IF reset THEN
	_bRetry := TRUE;
	Error 	:= FALSE;
	Aborted := FALSE;
END_IF

//============= State Control==================
IF NOT Execute THEN
	eSTATE:=STATE_RESETTING;
END_IF
IF Execute AND _bRetry AND NOT Robot._DI1.Error AND NOT Robot.Halt THEN
	PreviousStrStatus := strStatus;
	PreviousErrorCode := _UniqueErrorCode;
	uiExecutingStep   := uiResumeStep;
	Status := '';
	IF GVL_ADS.MachineState <>E_MachineState.Error THEN
		eSTATE:=STATE_EXECUTING;
	END_IF
END_IF
END_METHOD

METHOD  M_STATE_ABORTING
VAR_INPUT
END_VAR
CASE uiAbortingStep OF
	0 :
			
			tonTimeOut.IN 				:= FALSE;
			tonCheckRoundBeltDelay.IN	:= FALSE;
			_Abort := FALSE;
			_bRetry:= FALSE;
			IF strStatus = PreviousStrStatus THEN
				_UniqueErrorCode :=PreviousErrorCode;
			END_IF
			
			uiAbortingStep := 100;
    100:
			IF Robot._DI1.Error THEN
				uiAbortingStep := 200;
			ELSE
				uiAbortingStep := 9999;
			END_IF
	200:		
			 IF DAS_CoreSys.MachineControl.M_RobotResetCmd() THEN
				 uiAbortingStep := 300;
			 END_IF
	300:
			IF DAS_CoreSys.MachineControl.M_RobotStartCmd() THEN
				 uiAbortingStep := 400;
			 END_IF 
	400:
			IF Robot._DI1.Error THEN
		 		uiAbortingStep := 200;
			ELSE
				uiAbortingStep := 9999;
			END_IF
	9999:	
			_AbortCompleted:=TRUE;
END_CASE

IF _AbortCompleted THEN	
	eSTATE :=STATE_ABORTED;
END_IF
END_METHOD

METHOD  M_STATE_DONE
VAR_INPUT
END_VAR
Busy   := FALSE;
_Error := Error := FALSE;
_Abort := Abort := FALSE;
Done   := TRUE;

IF NOT Execute THEN
    eState := STATE_RESETTING;
END_IF
END_METHOD

METHOD  M_STATE_DORMANT
VAR_INPUT
END_VAR
// Clear FB output
Busy            := FALSE;
Done            := FALSE;
Aborted         := FALSE;
Error           := FALSE;
ErrorID         := 0;
Status          := '';
_ResetCompleted := FALSE;
_Error          := FALSE;
_Executed       := FALSE;

tonTimeOut.IN:=tonCheckRoundBeltDelay.IN:= FALSE;
strStatus :='FB_RobotRegionMove_RoundBelt: No Error';
uiExecutingStep :=uiResettingStep :=uiResumeStep :=0;
PreviousStrStatus			 :='';
PreviousErrorCode			 :='';
_bRetry			:= FALSE;
uiAbortingStep  := 0;
_AbortCompleted := FALSE;

// Wait Execute command
IF Execute AND NOT stop THEN
    eState := STATE_EXECUTING;
END_IF
END_METHOD

METHOD  M_STATE_ERROR
VAR_INPUT
END_VAR
ERROR   :=TRUE;
Busy	:=FALSE;
Status := strStatus;
UniqueErrorCode:=_UniqueErrorCode;
IF NOT Execute THEN	
eSTATE:=STATE_RESETTING;
END_IF
END_METHOD

METHOD  M_STATE_EXECUTING
VAR_INPUT
END_VAR
VAR_INST
	BoxReady_1st : BOOL;
	BoxReady_2nd : BOOL;
    uiBothStep : UINT;
    uiSingleClampStep : UINT;	
	Address_A : INT;
	Address_B : INT;
	A1Used	 : BOOL;
	A2Used	 : BOOL;
END_VAR
VAR
	
	
END_VAR
//20250418 note: current behavior : wait round belt finish rotating then check if box is ready , everything ready then call Robot start move
//				 Todo : consider if better call robot start move to waiting position and check box at same moment , Albert 

// Set Busy active edit by johnson
Busy := TRUE;
IF THIS^.Stop THEN // Pending the timeout when Stop signal occur
	tonTimeout.IN :=FALSE;
END_IF
// Service Process
CASE uiExecutingStep OF
	0:
        // Clear variable      
        uiBothStep := 0;
		uiSingleClampStep :=0;
		BoxReady_1st := 0;
		BoxReady_2nd := 0;
		tonTimeOut.IN:=FALSE;
		tonCheckRoundBeltDelay.IN :=FALSE;
        // Check command
        IF M_CheckCommand() THEN
            uiExecutingStep := 10;
		ELSE
			_Error:=TRUE;
        END_IF
    10:
        // Start process, check units first
        IF M_CheckUnitsReady() THEN
            uiExecutingStep := 20;
        END_IF
    20:
        // CHeck units not busy state
        IF M_CheckUnitsNotBusy() THEN
            uiExecutingStep := 30;
        END_IF
	30:
		IF M_CheckClampStatus() THEN
			uiExecutingStep := 1000;
		ELSE
			_Abort := TRUE;
		END_IF
   
	1000:   
			// Read   coordinate
			 Area := THIS^.Area;
 			 Address_A := LREAL_TO_INT(Info.A_Position);
			 Address_B := LREAL_TO_INT(Info.B_Position);
			 uiExecutingStep := 1100; 		
			 
	1100:
			// Check clamp userage
			IF UseA AND NOT UseB THEN
				//Only clampA
				A1Used := FALSE;
				A2Used := FALSE;
				uiExecutingStep := 10000;
			ELSIF NOT UseA AND UseB THEN
				//Only ClampB
				A1Used := FALSE;
				A2Used := FALSE;
				uiExecutingStep := 20000;
			ELSIF UseA AND UseB THEN
				//Both Clamps
				A1Used := TRUE;
				A2Used := TRUE;
				uiExecutingStep := 30000;
			END_IF
       
    10000: // Only ClampA 
        IF NOT Robot._DI1.Done THEN
			// Delay to make sure round belt is starting/finish rotating
			IF NOT RoundBelt.xBusy AND NOT RoundBelt.xError THEN
				tonCheckRoundBeltDelay.IN:=TRUE;
			ELSE
				tonCheckRoundBeltDelay.IN:=FALSE;	
			END_IF
		
		
		CASE uiSingleClampStep OF
			0:
				CASE Address_A OF						
							1: A1Used := TRUE;
							2: A2Used := TRUE;
				END_CASE
				
				IF tonCheckRoundBeltDelay.Q THEN
					 uiSingleClampStep:=50;  
				END_IF
				
			50:
				IF Get THEN  // Picking job , check box is ready
					IF A1Used AND Input.bRoundBelt_ChangeZoneA2Detect_Sensor =FALSE	THEN
						uiResettingStep := 10000;
						_Abort:=TRUE	;
						strStatus :='FB_RobotRegionMove_RoundBelt Step 10000: No Box on A1';
					ELSIF A2Used AND Input.bRoundBelt_ChangeZoneA3Detect_Sensor =FALSE	THEN
						uiResettingStep := 10000;
						_Abort:=TRUE	;
						strStatus :='FB_RobotRegionMove_RoundBelt Step 10000: No Box on A2';
					ELSE 
						uiSingleClampStep := 100;
					END_IF	
				ELSE		//Place job , check no box 
					IF A1Used AND Input.bRoundBelt_ChangeZoneA2Detect_Sensor =TRUE	THEN
						uiResettingStep := 10000;
						_Abort:=TRUE	;
						strStatus :='FB_RobotRegionMove_RoundBelt Step 10000: Box on A1';									
					ELSIF A2Used AND Input.bRoundBelt_ChangeZoneA3Detect_Sensor =TRUE	THEN
						uiResettingStep := 10000;
						_Abort:=TRUE	;
						strStatus :='FB_RobotRegionMove_RoundBelt Step 10000: Box on A2';
					ELSE
						uiSingleClampStep := 100;	
					END_IF				
				END_IF
	  
		  100 :  
		  		IF get THEN
					BoxReady_1st := (A1Used AND Input.bRoundBelt_ChangeZoneA2Detect_Sensor) OR
		  						 (A2Used AND Input.bRoundBelt_ChangeZoneA3Detect_Sensor);
				ELSE
					BoxReady_1st := (A1Used AND NOT Input.bRoundBelt_ChangeZoneA2Detect_Sensor) OR
		  						 (A2Used AND NOT Input.bRoundBelt_ChangeZoneA3Detect_Sensor);
				END_IF		
				IF BoxReady_1st THEN
					uiSingleClampStep:=9999;  
				END_IF			 
								 
		  9999:// 
	
		END_CASE				          		 
				  // Robot Abs move
           		 Robot.M_StartRobotAbsMove(GetBox:=Get,
											UseClampA:=UseA,
											UseClampB:=UseB,
											Area:=Area,
											ClampA_Address:=Address_A,
											ClampB_Address:=Address_B,
											BoxReady_1:=BoxReady_1st,
											BoxReady_2:=BoxReady_2nd);				  
		
        ELSE
			tonTimeOut.IN:=FALSE;
            uiExecutingStep := 10080;
        END_IF
			tonTimeOut.IN:=TRUE;
		IF tonTimeOut.Q=TRUE THEN
			uiResumeStep 	:= 10000;
			tonTimeOut.IN	:= FALSE;
			strStatus := 'FB_RobotRegionMove_RoundBelt Step 10000: Robot Abs Move timeout';
			_Abort			:= TRUE;
		END_IF	
		IF robot.Error THEN
			uiResumeStep 	:= 10000;
			tonTimeOut.IN	:= FALSE;
			_Abort 			:= TRUE;
			strStatus := CONCAT('FB_RobotRegionMove_RoundBlet Step 10000 : ',robot.ErrMsg);
		END_IF
    10080:
        Robot.M_ResetRobotAbsMove(UseA,UseB); // Clear command and go to place box
		tonTimeOut.IN:=TRUE;
        IF NOT Robot._DI1.Done THEN
			tonTimeOut.IN:=FALSE;
            uiExecutingStep := 99000; 
        END_IF
    	IF tonTimeOut.Q=TRUE THEN
			strStatus :='FB_RobotRegionMove_RoundBelt Step 10080: Reset Robot timeout';


			_Error:=TRUE;
		END_IF	
    
   20000: // Only ClampB
        IF NOT Robot._DI1.Done THEN
           IF NOT RoundBelt.xBusy AND NOT RoundBelt.xError THEN
				tonCheckRoundBeltDelay.IN:=TRUE;
			ELSE
				tonCheckRoundBeltDelay.IN:=FALSE;	
			END_IF
		
		
		CASE uiSingleClampStep OF
			0:
				CASE Address_B OF						
							1: A1Used := TRUE;
							2: A2Used := TRUE;
				END_CASE
				
				IF tonCheckRoundBeltDelay.Q THEN
					 uiSingleClampStep:=50;  
				END_IF
			
			50: 
				IF Get THEN  // Picking job , check box is ready
					IF A1Used AND Input.bRoundBelt_ChangeZoneA2Detect_Sensor =FALSE	THEN
						_Abort:=TRUE	;
						uiResettingStep := 20000;
						strStatus :='FB_RobotRegionMove_RoundBelt Step 20000: No Box on A1';		
					ELSIF A2Used AND Input.bRoundBelt_ChangeZoneA3Detect_Sensor =FALSE	THEN
						_Abort:=TRUE	;
						uiResettingStep := 20000;
						strStatus :='FB_RobotRegionMove_RoundBelt Step 20000: No Box on A2';
					ELSE
						uiSingleClampStep := 100;
					END_IF	
				ELSE		//Place job , check no box 
					IF A1Used AND Input.bRoundBelt_ChangeZoneA2Detect_Sensor =TRUE	THEN
						_Abort:=TRUE	;
						uiResettingStep := 20000;
						strStatus :='FB_RobotRegionMove_RoundBelt Step 20000: Box on A1';				
					ELSIF A2Used AND Input.bRoundBelt_ChangeZoneA3Detect_Sensor =TRUE	THEN
						_Abort:=TRUE	;
						uiResettingStep := 20000;
						strStatus :='FB_RobotRegionMove_RoundBelt Step 20000: Box on A2';
					ELSE
						uiSingleClampStep := 100;
					END_IF				
				END_IF
	  
		  100 :  
		  		IF get THEN
					BoxReady_2nd := (A1Used AND Input.bRoundBelt_ChangeZoneA2Detect_Sensor) OR
		  						 (A2Used AND Input.bRoundBelt_ChangeZoneA3Detect_Sensor);
				ELSE
					BoxReady_2nd := (A1Used AND NOT Input.bRoundBelt_ChangeZoneA2Detect_Sensor) OR
		  						 (A2Used AND NOT Input.bRoundBelt_ChangeZoneA3Detect_Sensor);
				END_IF		
				IF BoxReady_2nd THEN
					uiSingleClampStep:=9999;  
				END_IF			 
								 
		  9999:// 
	
		END_CASE				          		 
					  // Robot Abs move
           		 Robot.M_StartRobotAbsMove( GetBox:=Get,
											UseClampA:=UseA,
											UseClampB:=UseB,
											Area:=Area,
											ClampA_Address:=Address_A,
											ClampB_Address:=Address_B,
											BoxReady_1:=BoxReady_1st,
											BoxReady_2:=BoxReady_2nd);		  
		
        ELSE
			tonTimeOut.IN:=FALSE;
            uiExecutingStep := 20080;
        END_IF	
		tonTimeOut.IN:=TRUE;
		IF tonTimeOut.Q=TRUE THEN
			uiResumeStep 	:= 20000;
			tonTimeOut.IN	:= FALSE;
			strStatus := 'FB_RobotRegionMove_RoundBelt Step 20000: Robot Abs Move timeout';
			_Abort			:= TRUE;
		END_IF
		IF robot.Error THEN
			uiResumeStep := 20000;
			_Abort := TRUE;
			strStatus := CONCAT('FB_RobotRegionMove_RoundBlet Step 20000 : ',robot.ErrMsg);
		END_IF		          		 
			
       
		
    20080:
       Robot.M_ResetRobotAbsMove(UseA,UseB);; // Clear command
		tonTimeOut.IN:=TRUE;
        IF NOT Robot._DI1.Done THEN
			tonTimeOut.IN:=FALSE;
            uiExecutingStep := 99000;
        END_IF
		IF tonTimeOut.Q=TRUE THEN
			strStatus :='FB_RobotRegionMove_RoundBelt Step 20080: Reset Robot timeout';


			_Error:=TRUE;
		END_IF	
    30000: // Both Clamps
        	
			IF NOT RoundBelt.xBusy AND NOT RoundBelt.xError THEN
				tonCheckRoundBeltDelay.IN:=TRUE;
			ELSE
				tonCheckRoundBeltDelay.IN:=FALSE;	
			END_IF
		
		  CASE uiBothStep OF
           		0://	
					BoxReady_1st := FALSE;
					BoxReady_2nd := FALSE;
					
					IF tonCheckRoundBeltDelay.Q THEN
						uiBothStep:=100;	
					END_IF
				100:
					IF Get THEN  // Picking job , check box is ready
						IF  Input.bRoundBelt_ChangeZoneA2Detect_Sensor =FALSE	THEN
							_Abort:=TRUE	;
							uiResettingStep := 30000;
							strStatus :='FB_RobotRegionMove_RoundBelt Step 30000: No Box on A1';
						END_IF				
						IF  Input.bRoundBelt_ChangeZoneA3Detect_Sensor =FALSE	THEN
							_Abort:=TRUE	;
							uiResettingStep := 30000;
							strStatus :='FB_RobotRegionMove_RoundBelt Step 30000: No Box on A2';
						END_IF	
					ELSE		//Place job , check no box 
						IF  Input.bRoundBelt_ChangeZoneA2Detect_Sensor =TRUE	THEN
							_Abort:=TRUE	;
							uiResettingStep := 30000;
							strStatus :='FB_RobotRegionMove_RoundBelt Step 30000: Box on A1';
						END_IF				
						IF  Input.bRoundBelt_ChangeZoneA3Detect_Sensor =TRUE	THEN
							_Abort:=TRUE	;
							uiResettingStep := 30000;
							strStatus :='FB_RobotRegionMove_RoundBelt Step 30000: Box on A2';
						END_IF				
					END_IF
					IF NOT _Error THEN
						uiBothStep:=1000;
					END_IF
				1000:	
						
						BoxReady_1st :=TRUE;
						uiBothStep:=2000;
					
						
				2000:					
						IF Robot._DI1.Notification THEN
							uiBothStep:=3000;
						END_IF
				3000:	
						 BoxReady_2nd :=TRUE;						 
					     uiBothStep:=9999;
				
				9999: //Wait		
        // wait reset
        END_CASE

       	  // Robot Abs move
           		 Robot.M_StartRobotAbsMove( GetBox:=Get,
											UseClampA:=UseA,
											UseClampB:=UseB,
											Area:=Area,
											ClampA_Address:=Address_A,
											ClampB_Address:=Address_B,
											BoxReady_1:=BoxReady_1st,
											BoxReady_2:=BoxReady_2nd);	
		
		
        IF Robot._DI1.Done THEN
			tonTimeOut.IN:=FALSE;
            uiExecutingStep := 30080;
        END_IF
		tonTimeOut.IN:=TRUE;
		IF tonTimeOut.Q=TRUE THEN
			uiResumeStep 	:= 30000;
			tonTimeOut.IN	:= FALSE;
			strStatus := 'FB_RobotRegionMove_RoundBelt Step 30000: Robot Abs Move timeout';
			_Abort			:= TRUE;
		END_IF
		IF robot.Error THEN
			uiResumeStep := 30000;
			_Abort := TRUE;
			strStatus := CONCAT('FB_RobotRegionMove_RoundBlet Step 30000 : ',Robot.ErrMsg);
		END_IF	
		
    30080: // Check robot command is clear
        
        Robot.M_ResetRobotAbsMove(UseA,UseB);

        IF NOT Robot._DI1.Done THEN
			tonTimeOut.IN:=FALSE;
            uiExecutingStep := 99000; // go to place step
        END_IF    
   		tonTimeOut.IN:=TRUE;
		IF tonTimeOut.Q=TRUE THEN
			strStatus :='FB_RobotRegionMove_RoundBelt Step 30080: Stop Robot timeout';




			_Error:=TRUE;
		END_IF	
   
    99000:
			IF Get THEN  // Picking job , check box putted
				IF A1Used AND Input.bRoundBelt_ChangeZoneA2Detect_Sensor =TRUE	THEN
					_Error:=TRUE	;
					strStatus :='FB_RobotRegionMove_RoundBelt Step 99000: Box still on A1';


				END_IF				
				IF A2Used AND Input.bRoundBelt_ChangeZoneA3Detect_Sensor =TRUE	THEN
					_Error:=TRUE	;
					strStatus :='FB_RobotRegionMove_RoundBelt Step 99000: Box still on A2';


				END_IF	
			ELSE		//Place job , check no box 
				IF A1Used AND Input.bRoundBelt_ChangeZoneA2Detect_Sensor =FALSE	THEN
					_Error:=TRUE	;
					strStatus :='FB_RobotRegionMove_RoundBelt Step 99000: No Box on A1';


				END_IF				
				IF A2Used AND Input.bRoundBelt_ChangeZoneA3Detect_Sensor =FALSE	THEN
					_Error:=TRUE	;
					strStatus :='FB_RobotRegionMove_RoundBelt Step 99000: No Box on A2';


				END_IF	
			
			END_IF
			IF NOT _Error THEN
			 	uiExecutingStep := 99100;
			 END_IF
	99100: // process done
                Status    := 'FB_RobotRegionMove_RoundBelt Step 99100: Process completed';
        	_Executed := TRUE;
END_CASE

// ==================== STATE Control ========================
IF NOT Execute THEN
    eState 	:= STATE_RESETTING;
ELSIF _Error THEN
    eState 	:= STATE_ERROR;
ELSIF _Abort THEN
	eSTATE	:= STATE_ABORTING;
ELSIF _Executed THEN
    eState 	:= STATE_DONE;
END_IF
END_METHOD

METHOD  M_STATE_RESETTING
VAR_INPUT
END_VAR
// Done := false 更改到Dormant 清除確保，上位檢查到done 後可以直接下Execute

CASE uiResettingStep OF

	0:
		tonTimeOut.IN:=FALSE;
		Robot.M_ResetAllCommand();
		Robot.M_ResetRobotAbsMove(TRUE,TRUE);
		uiResettingStep:=100;

	100:

		uiResettingStep:=9999;
		
	9999:
//		Done := FALSE;
//		Busy := FALSE;
		_ResetCompleted:=TRUE;
END_CASE
IF _ResetCompleted THEN
	eSTATE:=STATE_DORMANT;
END_IF
END_METHOD

END_FUNCTION_BLOCK

// ---- Library/20_MachineUnits/21_StorageArea/Service_Robot/FB_RobotAbsMove_V2.TcPOU
// Jidien Kachu Edited in 2025/10/14
FUNCTION_BLOCK FB_RobotAbsMove_V2 EXTENDS FB_ObjectBase_V2 IMPLEMENTS IBasicElement
VAR_INPUT
    Robot         				: REFERENCE TO FB_FanucRobot_Basic_V2;
    LowerConveyor 				: REFERENCE TO FB_Motor;
    // Command   : ST_WareHouseWithRobotMove_Command;
    Info 						: st_AutoSixAxisAbsMoveParameter;
	Input 						: ST_InputTable;
    Stop 						: BOOL;
	Output 						: ST_OutputTable;
	Cylinder 					: REFERENCE TO UNI_CylinderList;
	bCheckUpperCV_ServiceDone	: BOOL;
END_VAR
VAR_OUTPUT
    // Status : ST_WareHouseWithRobotMove_Status;
	AClampMoveDone	: BOOL;
	BClampMoveDone	: BOOL;
END_VAR
VAR
    //_Abort       : BOOL;
    strStatus    : STRING;
    uiResumeStep : UINT;

    Area : E_RobotArea;
    UseA : BOOL;
    UseB : BOOL;

    Get                         : BOOL;
    tonTimeOut                  : TON;
	bTimeOutIN					: BOOL;
	tonDelay					 : TON;
    _UniqueErrorCode            : STRING;
    FirstSensorOfLowerConveyor  : BOOL;
    SecondSensorOfLowerConveyor : BOOL;

	//Added by Jidien Kachu in 2025/10/09
	uiLastBothStep	: UINT;
	uiLastSingleClampStep	: UINT;
	bRobotTimeOutIN	: BOOL;
	tonRobotTimeOut	: TON;
	uiBothStep	: UINT;
	uiSingleClampStep	: UINT;
	bMotorDelayIN	: BOOL;
	tonMotorDelay	: TON;
	bIOTimeoutIN	: BOOL;
	tonIOTimeout	: TON;
	bRetry: BOOL;
	
	//Added by Gamin in 2025//11/24
	_AClampDoingWork	: BOOL;
	_BClampDoingWork	: BOOL;
END_VAR

SUPER^.A10_StateControl();
A00_BasicUnits();
FirstSensorOfLowerConveyor := Input.bLowCV_BoxArrived_Sensor;
SecondSensorOfLowerConveyor := NOT Input.bLowCV_2ndBoxGap_Sensor;// .bLowCV_Block2Detect_Sensor;

(*============================================================
Create Date : 2025/11/22
Last Update	: 2026/04/01
Change Log  : 2025/11/24，send flag A clamp done and B clamp done for C# use to SQL // Edited : Gamin
			  2026/04/01，移植泰興鏡射機版本。
============================================================*)

ACTION A00_BasicUnits:
tonTimeOut(IN:= bTimeOutIN AND NOT THIS^.Stop, PT:=T#60S);
tonDelay(PT:=T#1S);
ErrorID :=2200;
tonMotorDelay(IN:= bMotorDelayIN,PT:=T#1S);
tonIOTimeout(IN:= bIOTimeoutIN,PT:= T#1S);
END_ACTION

METHOD M_CheckClampStatus : BOOL
VAR_INPUT
END_VAR
M_CheckClampStatus := FALSE;

IF NOT UseA AND NOT UseB THEN
	M_CheckClampStatus 	:= FALSE;
	strStatus 			:= 'FB_RobotAbsMove_V2: Wrong Command , Both Clammp not used';
	RETURN;
END_IF

IF UseA THEN
	IF Get THEN
		IF NOT Robot._DI1.ClampA_Open THEN
			M_CheckClampStatus  := FALSE;
			strStatus			:= 'FB_RobotAbsMove_V2: Robot Use A Clamp Get ,but Clamp not open ';
			RETURN;
		END_IF
	ELSE
		IF Robot._DI1.ClampA_Open THEN
			M_CheckClampStatus	:= FALSE;
			strStatus			:= 'FB_RobotAbsMove_V2: Robot Use A Clamp Place ,but Clamp open';
			RETURN;
		END_IF
	END_IF
END_IF
IF UseB THEN
	IF Get THEN
		IF NOT Robot._DI1.ClampB_Open THEN
			M_CheckClampStatus  := FALSE;
			strStatus			:= 'FB_RobotAbsMove_V2: Robot Use B Clamp Get ,but Clamp not open ';
			RETURN;
		END_IF
	ELSE
		IF Robot._DI1.ClampB_Open THEN
			M_CheckClampStatus	:= FALSE;
			strStatus			:= 'FB_RobotAbsMove_V2: Robot Use B Clamp Place ,but Clamp open';
			RETURN;
		END_IF
	END_IF
END_IF

M_CheckClampStatus := TRUE;
END_METHOD

METHOD M_CheckCommand : BOOL // True : Command is useful
VAR_INPUT
END_VAR
VAR
	
END_VAR
// Check command paremeter is correct


IF Info.A_Get <> Info.B_Get THEN
	strStatus:='FB_RobotAbsMove_V2: Wrong command ,GetA not match to GetB';
	M_CheckCommand:=FALSE;
	RETURN;
ELSE		
	THIS^.Get :=Info.A_Get;
END_IF

IF Info.A_Area<> Info.B_Area THEN
	IF NOT(Info.A_Area=99 OR Info.B_Area=99) THEN
	strStatus:='FB_RobotAbsMove_V2: Wrong command ,Area A not match to Area B';
	M_CheckCommand:=FALSE;
	RETURN;
END_IF
END_IF

IF Info.A_Area = 99 AND Info.B_Area = 99 THEN
	strStatus:='FB_RobotAbsMove_V2: Wrong command ,Both Area are 99';
	M_CheckCommand:=FALSE;
	RETURN;
END_IF

CASE LREAL_TO_INT(Info.A_Area) OF
	1 : //Normal command : RoundBelt
		IF Info.A_Position<1 OR  Info.A_Position>3 THEN
			strStatus:='FB_RobotAbsMove_V2: Wrong command ,Position A Not allow';
			M_CheckCommand:=FALSE;
			RETURN;	
		ELSE
			Area := E_RobotArea.RoundBelt;
			UseA :=TRUE	;	
		END_IF
		
	2:	//Buffer area
		IF Info.A_Position<1 OR  Info.A_Position>40 THEN
			strStatus:='FB_RobotAbsMove_V2: Wrong command ,Position A Not allow';
			M_CheckCommand:=FALSE;
			RETURN;	
		ELSE
			Area := E_RobotArea.BufferArea;
			UseA :=TRUE	;	
		END_IF
	3: //Allocated/Empty conveyor
		IF Info.A_Position<1 OR  Info.A_Position>2 THEN
			strStatus:='FB_RobotAbsMove_V2: Wrong command ,Position A Not allow';
			M_CheckCommand:=FALSE;
			RETURN;	
		ELSE
			Area := E_RobotArea.TransmitCV;
			UseA :=TRUE	;	
		END_IF
	5: //FeedIn/Out conveyor
		IF Info.A_Position<1 OR  Info.A_Position>5 THEN
			strStatus:='FB_RobotAbsMove_V2: Wrong command ,Position A Not allow';
			M_CheckCommand:=FALSE;
			RETURN;	
		ELSIF Info.A_Position=3 AND Get THEN
			strStatus:='FB_RobotAbsMove_V2: Wrong command ,Can Not Get box from FeedOut conveyor ';
			M_CheckCommand:=FALSE;
			RETURN;	
		ELSE
			Area := E_RobotArea.InOutConveyor;
			UseA :=TRUE	;	
		END_IF
	7: // PullOut conveyor
		IF Info.A_Position<1 OR  Info.A_Position>2 THEN
			strStatus:='FB_RobotAbsMove_V2: Wrong command ,Position A Not allow';
			M_CheckCommand:=FALSE;
			RETURN;	
		ELSE
			Area := E_RobotArea.PullOutConveyor;
			UseA :=TRUE	;	
		END_IF
	
	99: //ClampA not use
		UseA :=FALSE;
	
	ELSE //Wrong command
		strStatus:='FB_RobotAbsMove_V2: Wrong command ,Area_A not allow ';
		M_CheckCommand:=FALSE;
		RETURN;

END_CASE

CASE LREAL_TO_INT(Info.B_Area) OF
	1 : //Normal command : RoundBelt
		IF Info.B_Position<1 OR  Info.B_Position>3 THEN
			strStatus:='FB_RobotAbsMove_V2: Wrong command ,Position B Not allow';
			M_CheckCommand:=FALSE;
			RETURN;	
		ELSE
			Area := E_RobotArea.RoundBelt;
			UseB :=TRUE	;	
		END_IF
		
	2:	
		IF Info.B_Position<1 OR  Info.B_Position>40 THEN
			strStatus:='FB_RobotAbsMove_V2: Wrong command ,Position B Not allow';
			M_CheckCommand:=FALSE;
			RETURN;	
		ELSE
			Area := E_RobotArea.BufferArea;
			UseB :=TRUE	;	
		END_IF
	3:
		IF Info.B_Position<1 OR  Info.B_Position>2 THEN
			strStatus:='FB_RobotAbsMove_V2: Wrong command ,Position B Not allow';
			M_CheckCommand:=FALSE;
			RETURN;	
		ELSE
			Area := E_RobotArea.TransmitCV;
			UseB :=TRUE	;	
		END_IF
	5:
		IF Info.B_Position<1 OR  Info.B_Position>5 THEN
			strStatus:='FB_RobotAbsMove_V2: Wrong command ,Position B Not allow';
			M_CheckCommand:=FALSE;
			RETURN;	
		ELSE
			Area := E_RobotArea.InOutConveyor;
			UseB :=TRUE	;	
		END_IF
	7:
		IF Info.B_Position<1 OR  Info.B_Position>2 THEN
			strStatus:='FB_RobotAbsMove_V2: Wrong command ,Position B Not allow';
			M_CheckCommand:=FALSE;
			RETURN;	
		ELSIF Info.B_Position=3 AND Get THEN
			strStatus:='FB_RobotAbsMove_V2: Wrong command ,Can Not Get box from FeedOut conveyor ';
			M_CheckCommand:=FALSE;
			RETURN;	
		ELSE
			Area := E_RobotArea.PullOutConveyor;
			UseB :=TRUE	;	
		END_IF
	
	99: //ClampA not use
		UseB :=FALSE;
	
	ELSE //Wrong command
		strStatus:='FB_RobotAbsMove_V2: Wrong command ,Area_B not allow ';
		M_CheckCommand:=FALSE;
		RETURN;

END_CASE


M_CheckCommand:=TRUE;
END_METHOD

METHOD M_CheckUnitsNotBusy : BOOL
VAR_INPUT
END_VAR
M_CheckUnitsNotBusy := true;
END_METHOD

METHOD M_CheckUnitsReady : BOOL
VAR_INPUT
END_VAR
M_CheckUnitsReady := true;
END_METHOD

METHOD  M_STATE_ABORTED
VAR_INPUT
END_VAR

//Edited by Jidien Kachu in 2025/10/28
IF NOT bRetry THEN
	ERROR :=TRUE;
	Busy    := FALSE;
	Aborted := TRUE;
	Status := strStatus;
	UniqueErrorCode:=_UniqueErrorCode;
	uiAbortingStep := 0;
	_AbortCompleted:=FALSE;//Edited by Jidien Kachu in 2025/10/14
END_IF

IF Reset THEN
	bRetry := TRUE;
	ERROR :=FALSE;
	Aborted := FALSE;
END_IF
IF NOT Execute THEN
	eSTATE:=STATE_RESETTING;
END_IF

IF Execute AND bRetry AND NOT Robot.Error AND NOT Robot.Halt THEN
	uiExecutingStep :=uiResumeStep;

	//Edited by Jidien Kachu in 2025/10/14
	uiBothStep := uiLastBothStep;
	uiSingleClampStep := uiLastSingleClampStep;
	Status := '';


	//////////////////////////////////////
	IF GVL_ADS.MachineState <>E_MachineState.Error THEN
		eSTATE:=STATE_EXECUTING;
	END_IF
END_IF
END_METHOD

METHOD  M_STATE_ABORTING
VAR_INPUT
END_VAR
CASE uiAbortingStep OF
	0 :
			tonDelay.IN 	   := FALSE;
			bTimeOutIN  	   := FALSE;
			tonRobotTimeOut.IN := FALSE;
			_Abort 			   := FALSE;
			bRetry			   := FALSE;
			//Edited by Jidien Kachu in 2025/10/14
			LowerConveyor.M_MotorStop();
			IF 	LowerConveyor.InStopped THEN
				uiAbortingStep:=100;
			END_IF
    100:
			IF Robot._DI1.Error THEN
				uiAbortingStep := 200;
			ELSE
				uiAbortingStep := 9999;
			END_IF
	200:		
			 IF DAS_CoreSys.MachineControl.M_RobotResetCmd() THEN
				 uiAbortingStep := 300;
			 END_IF
	300:
			IF DAS_CoreSys.MachineControl.M_RobotStartCmd() THEN
				 uiAbortingStep := 400;
			 END_IF 
	400:
			IF Robot._DI1.Error THEN
		 		uiAbortingStep := 200;
			ELSE
				uiAbortingStep := 9999;
			END_IF
	
	9999:	
			_AbortCompleted:=TRUE;
END_CASE

IF _AbortCompleted THEN	
	eSTATE :=STATE_ABORTED;
END_IF
END_METHOD

METHOD  M_STATE_DONE
VAR_INPUT
END_VAR
Busy   := FALSE;
_Error := Error := FALSE;
_Abort := Abort := FALSE;
Done   := TRUE;

IF NOT Execute THEN
    eState := STATE_RESETTING;
END_IF
END_METHOD

METHOD  M_STATE_DORMANT
VAR_INPUT
END_VAR
// Clear FB output
Busy            := FALSE;
Done            := FALSE;
Aborted         := FALSE;
Error           := FALSE;
ErrorID         := 0;
Status          := '';
_ResetCompleted := FALSE;
_AbortCompleted := FALSE;
_Error          := FALSE;
_Executed       := FALSE;
tonDelay.IN := FALSE	;
bTimeOutIN:=FALSE;
strStatus :='FB_RobotAbsMove_V2: No Error';
uiExecutingStep :=uiResettingStep :=uiResumeStep :=0;
AClampMoveDone	:= FALSE;
BClampMoveDone	:= FALSE;
_AClampDoingWork	:= FALSE;
_BClampDoingWork	:= FALSE;
bRetry := FALSE;
uiBothStep := 0;
uiSingleClampStep :=0;

// Wait Execute command
IF Execute AND NOT stop THEN
    eState := STATE_EXECUTING;
END_IF
END_METHOD

METHOD  M_STATE_ERROR
VAR_INPUT
END_VAR
ERROR   :=TRUE;
Busy	:=FALSE;
Status := strStatus;
UniqueErrorCode:=_UniqueErrorCode;
ErrorID :=2200;

IF NOT Execute THEN	
	eSTATE:=STATE_RESETTING;
END_IF
END_METHOD

METHOD  M_STATE_EXECUTING
VAR_INPUT
END_VAR
VAR_INST
    ActionMode       : E_ReloadRoundBoxAction;
	BoxReady_1st : BOOL;
	BoxReady_2nd : BOOL;
    CarrierReady_1st : BOOL;
    CarrierReady_2nd : BOOL;
    //uiBothStep : UINT;
    //uiSingleClampStep : UINT;	
	Area : E_RobotArea;
	Address_A : INT;
	Address_B : INT;
END_VAR
VAR
	WareHouse: INT;
END_VAR
// Set Busy active edit by johnson
Busy := TRUE;
(*IF THIS^.Stop THEN // Pending the timeout when Stop signal occur
	tonTimeout.IN :=FALSE;
END_IF*)
// Service Process
CASE uiExecutingStep OF
	0:
        // Clear variable
        ActionMode       := E_ReloadRoundBoxAction.Undefined;
        CarrierReady_1st := FALSE;
        CarrierReady_2nd := FALSE;
        uiBothStep := 0;
		uiSingleClampStep :=0;
		uiLastBothStep := 0;//Edited by Jidien Kachu in 2025/10/14
		uiLastSingleClampStep := 0;//Edited by Jidien Kachu in 2025/10/14
		BoxReady_1st := FALSE;
		BoxReady_2nd := FALSE;
		bTimeOutIN:=FALSE;
        // Check command
        IF M_CheckCommand() THEN
            uiExecutingStep := 10;
		ELSE
			_Error:=TRUE;
        END_IF
    10:
        // Start process, check units first
        IF M_CheckUnitsReady() THEN
            uiExecutingStep := 20;
        END_IF
    20:
        // CHeck units not busy state
        IF M_CheckUnitsNotBusy() THEN
            uiExecutingStep := 30;
        END_IF
	30:
		IF M_CheckClampStatus() THEN
            uiExecutingStep := 1000;
		ELSE
			_Abort := TRUE;
        END_IF
   
	1000:   
			// Read   coordinate
			 Area := THIS^.Area;
 			 Address_A := LREAL_TO_INT(Info.A_Position);
			 Address_B := LREAL_TO_INT(Info.B_Position);
			 
			IF UseA AND NOT UseB THEN
				//Only clampA
				uiExecutingStep := 10000;
			ELSIF NOT UseA AND UseB THEN
				//Only ClampB 
				uiExecutingStep := 20000;
			ELSIF UseA AND UseB THEN
				//Both Clamps
				uiExecutingStep := 30000;		
			END_IF
       
    10000: // Only ClampA 
        IF NOT Robot._DI1.Done THEN
            //Edited by Jidien Kachu in 2025/10/14
				CASE uiSingleClampStep OF
					0://
						IF Area= E_RobotArea.InOutConveyor AND Address_A=3 THEN
							IF Cylinder.List.fbLowCV_Block1.InRearPosition THEN
								uiSingleClampStep:=100;// Need to control feedout conveyor
							ELSE
								_Error := TRUE;
								strStatus := 'FB_RobotAbsMove_V2 Step 10000: Block 2 cylinder inrearPosition';
							END_IF
						ELSE
							uiSingleClampStep:=1000;	
						END_IF
					100:	
						tonDelay.IN := FALSE	;
						LowerConveyor.M_MoveBackward();
						IF (NOT FirstSensorOfLowerConveyor) AND (NOT SecondSensorOfLowerConveyor) THEN
							bTimeOutIN:=FALSE;;
							uiSingleClampStep:=150;
						END_IF
						bTimeOutIN:=TRUE;
						//Edited by Jidien Kachu in 2025/10/14
						IF tonTimeOut.Q=TRUE OR robot._DI1.Error THEN
							strStatus :='FB_RobotAbsMove_V2 Step 10000: Empty Conveyor timeout';
	//						_Error:=TRUE;
							_Abort := TRUE;
							uiLastSingleClampStep := 0;
							uiResumeStep := 10000;
							uiAbortingStep := 0;
						END_IF
						//////////////////////////////////////////
					150:
						tonDelay.IN := TRUE;
						IF tonDelay.Q THEN
							uiSingleClampStep:=200;
						END_IF	
					200:
						tonDelay.IN := FALSE	;
						LowerConveyor.M_MotorStop();
						uiSingleClampStep:=300;
					
					300:
						IF 	LowerConveyor.InStopped THEN
							bTimeOutIN:=FALSE;
							BoxReady_1st:=TRUE;
							uiSingleClampStep:=9999;
						END_IF
						bTimeOutIN:=TRUE;
						//Edited by Jidien Kachu in 2025/10/14
						IF tonTimeOut.Q=TRUE OR Robot._DI1.Error THEN
							strStatus :='FB_RobotAbsMove_V2 Step 10000: Stop Conveyor timeout';
	//						_Error:=TRUE;
							_Abort := TRUE;
							uiLastSingleClampStep := 200;
							uiResumeStep := 10000;
							uiAbortingStep := 0;
						END_IF	
						//////////////////////////////////////////
					1000:
						// 檢查 A爪去夾爪時，要確保上層輸送帶是完成的。
							IF Area= E_RobotArea.InOutConveyor AND Address_A = 2 THEN
								IF bCheckUpperCV_ServiceDone THEN
									BoxReady_1st:=TRUE;
									_AClampDoingWork := TRUE;
									uiSingleClampStep:=9999;
								END_IF
							ELSE
							BoxReady_1st:=TRUE;
							_AClampDoingWork := TRUE;
							uiSingleClampStep:=9999;
							END_IF
					9999: //Wait	
				END_CASE
//			END_IF
			
			          		 
				  // Robot Abs move
           		 Robot.M_StartRobotAbsMove(GetBox:=Get,
											UseClampA:=UseA,
											UseClampB:=UseB,
											Area:=Area,
											ClampA_Address:=Address_A,
											ClampB_Address:=Address_B,
											BoxReady_1:=BoxReady_1st,
											BoxReady_2:=BoxReady_2nd);		

			// robot doing AClamp done
			IF Get THEN
				IF _AClampDoingWork AND NOT Robot._DI1.ClampA_Open THEN
					AClampMoveDone := TRUE;
				END_IF
			ELSE
				IF _AClampDoingWork AND Robot._DI1.ClampA_Open THEN
					AClampMoveDone := TRUE;
				END_IF
			END_IF	  
		
        ELSE
            uiExecutingStep := 10080;
        END_IF
		IF tonRobotTimeOut.Q THEN
			_Abort 		 := TRUE;
			uiResumeStep := 10000;
			strStatus 	 := 'FB_RobotAbsMove_V2 Step 10000: Robot Move timeout';
		END_IF
		IF Robot._DI1.Error THEN
			_Abort		:= TRUE;
			uiResumeStep:= 10000;
			strStatus	:= CONCAT(STR1 := 'FB_RobotAbsMove_V2 Step 10000:',
								  STR2 := Robot.ErrMsg);
        END_IF
		
    10080:
        Robot.M_ResetRobotAbsMove(UseA,UseB); // Clear command and go to place box
		bTimeOutIN:=TRUE;
        IF NOT Robot._DI1.Done THEN
			bTimeOutIN:=FALSE;
            uiExecutingStep := 40000; 
        END_IF
    	IF tonTimeOut.Q=TRUE THEN
			strStatus :='FB_RobotAbsMove_V2 Step 10080: Reset Robot timeout';
			_Error:=TRUE;
		END_IF
		
    
   20000: // Only ClampB
        IF NOT Robot._DI1.Done THEN
				CASE uiSingleClampStep OF
					0://
						IF Area= E_RobotArea.InOutConveyor AND Address_B=3 THEN
							IF Cylinder.List.fbLowCV_Block1.InRearPosition THEN
								uiSingleClampStep:=100;// Need to control feedout conveyor
							ELSE
								_Error := TRUE;
								strStatus := 'FB_RobotAbsMove_V2 Step 20000: Block 2 cylinder inrearPosition';
							END_IF
						ELSE
							uiSingleClampStep:=1000;	
						END_IF
					100:	
						tonDelay.IN := FALSE;
						LowerConveyor.M_MoveBackward();
						IF (NOT FirstSensorOfLowerConveyor) AND (NOT SecondSensorOfLowerConveyor) THEN
							bTimeOutIN:=FALSE;
							uiSingleClampStep:=150;
						END_IF
						bTimeOutIN:=TRUE;
						//Edited by Jidien Kachu in 2025/10/14
						IF tonTimeOut.Q=TRUE OR Robot._DI1.Error THEN
							strStatus :='FB_RobotAbsMove_V2 Step 20000: Empty Conveyor timeout';
							_Abort := TRUE;
							uiLastSingleClampStep := 0;
							uiResumeStep := 20000;
							uiAbortingStep := 0;
						END_IF	
						///////////////////////////////////////////
					150:
						tonDelay.IN := TRUE;
						IF tonDelay.Q THEN
							uiSingleClampStep:=200;
						END_IF	
		
					200:
						tonDelay.IN := FALSE;
						LowerConveyor.M_MotorStop();
						uiSingleClampStep:=300;
					
					300:
						IF 	LowerConveyor.InStopped THEN
							bTimeOutIN:=FALSE;
							BoxReady_2nd:=TRUE;
							uiSingleClampStep:=9999;
						END_IF
						bTimeOutIN:=TRUE;
						//Edited by Jidien Kachu in 2025/10/14
						IF tonTimeOut.Q=TRUE OR Robot._DI1.Error THEN
							strStatus := 'FB_RobotAbsMove_V2 Step 20000: Stop Conveyor timeout';
	//						_Error:=TRUE;
							_Abort := TRUE;
							uiLastSingleClampStep := 200;
							uiResumeStep := 20000;
							uiAbortingStep := 0;
						END_IF	
						///////////////////////////////////////////
					1000:
							// 檢查 A爪去夾爪時，要確保上層輸送帶是完成的。
							IF Area= E_RobotArea.InOutConveyor AND Address_B = 1 THEN
								IF bCheckUpperCV_ServiceDone THEN
									BoxReady_2nd	 := TRUE;
									_BClampDoingWork := TRUE;
									uiSingleClampStep:=9999;
								END_IF
							ELSE
							BoxReady_2nd	 := TRUE;
							_BClampDoingWork := TRUE;
							uiSingleClampStep:=9999;
							END_IF

					
					9999: //Wait			
				END_CASE
//			END_IF
			
			          		 
				  // Robot Abs move
           		 Robot.M_StartRobotAbsMove( GetBox:=Get,
											UseClampA:=UseA,
											UseClampB:=UseB,
											Area:=Area,
											ClampA_Address:=Address_A,
											ClampB_Address:=Address_B,
											BoxReady_1:=BoxReady_1st,
											BoxReady_2:=BoxReady_2nd);	
											
			// robot doing BClamp done
			IF Get THEN
				IF _BClampDoingWork AND NOT Robot._DI1.ClampB_Open THEN 
					BClampMoveDone := TRUE;
				END_IF
			ELSE
				IF _BClampDoingWork AND  Robot._DI1.ClampB_Open THEN 
					BClampMoveDone := TRUE;
				END_IF
			END_IF
											
        ELSE
            uiExecutingStep := 20080;
        END_IF
		IF tonRobotTimeOut.Q THEN
			_Abort 		 := TRUE;
			uiResumeStep := 20000;
			strStatus 	 := 'FB_RobotAbsMove_V2 Step 20000: Robot Move timeout';
		END_IF
		IF Robot._DI1.Error THEN
			_Abort		:= TRUE;
			uiResumeStep:= 20000;
			strStatus	:= CONCAT(STR1 := 'FB_RobotAbsMove_V2 Step 20000:',
								  STR2 := Robot.ErrMsg);
        END_IF
		
    20080:
       Robot.M_ResetRobotAbsMove(UseA,UseB); // Clear command 
        IF NOT Robot._DI1.Done THEN
            uiExecutingStep := 40000; 
        END_IF
		bTimeOutIN:=TRUE;
		IF tonTimeOut.Q=TRUE THEN
			strStatus :='FB_RobotAbsMove_V2 Step 20080: Reset Robot timeout';
			_Error:=TRUE;
		END_IF	
    30000: // Both Clamps
			CASE uiBothStep OF
           		0://	
					BoxReady_1st := FALSE;
					BoxReady_2nd := FALSE;
					IF Area= E_RobotArea.InOutConveyor AND Address_A=3 THEN
						IF Cylinder.List.fbLowCV_Block1.InRearPosition THEN
								uiBothStep:=100;// Need to control feedout conveyor
							ELSE
								_Error := TRUE;
								strStatus := 'FB_RobotAbsMove_V2 Step 30000: Block 1 cylinder inrearPosition';
							END_IF
					ELSE
						uiBothStep:=1000;	
					END_IF
				100:	
					tonDelay.IN := FALSE;
					LowerConveyor.M_MoveBackward();
					bTimeOutIN:=FALSE;
					IF (NOT FirstSensorOfLowerConveyor) AND (NOT SecondSensorOfLowerConveyor) THEN
						uiBothStep:=150;
					END_IF
					bTimeOutIN:=TRUE;
					//Edited by Jidien Kachu in 2025/10/14
					IF tonTimeOut.Q=TRUE OR Robot._DI1.Error THEN
						strStatus :='FB_RobotAbsMove_V2 Step 30000: Empty Robot timeout';
//						_Error:=TRUE;
						_Abort := TRUE;
						uiLastBothStep := 0;
						uiResumeStep := 30000;
						uiAbortingStep := 0;
					END_IF	
					///////////////////////////////////////////					
				150:
					tonDelay.IN := TRUE;
					IF tonDelay.Q THEN
						uiBothStep:=200;
					END_IF	
				
				200:
					tonDelay.IN := FALSE;
					LowerConveyor.M_MotorStop();
					uiBothStep:=300;
				
				300:
					IF 	LowerConveyor.InStopped THEN
						bTimeOutIN:=FALSE;
						BoxReady_1st:=TRUE;
						uiBothStep:=2000;
					END_IF
					bTimeOutIN:=TRUE;
					//Edited by Jidien Kachu in 2025/10/14
					IF tonTimeOut.Q=TRUE OR Robot._DI1.Error THEN
						strStatus :='FB_RobotAbsMove_V2 Step 30000: Stop Robot timeout';
//						_Error:=TRUE;
						_Abort := TRUE;
						uiLastBothStep := 200;
						uiResumeStep := 30000;
						uiAbortingStep := 0;
					END_IF	
					///////////////////////////////////////////					
				1000:
						// 檢查 A爪去夾爪時，要確保上層輸送帶是完成的。
						IF Area= E_RobotArea.InOutConveyor AND Address_A = 2 THEN
							IF bCheckUpperCV_ServiceDone THEN
						BoxReady_1st	 := TRUE;
						_AClampDoingWork := TRUE;
								uiBothStep		 := 2000;
							END_IF
						ELSE
							BoxReady_1st	 := TRUE;
							_AClampDoingWork := TRUE;
							uiBothStep		 := 2000;
						END_IF
						
				2000:
						IF Robot._DI1.Notification THEN
							uiBothStep:=3000;
						END_IF
						//Edited by Jidien Kachu in 2025/10/14
						IF Robot._DI1.Error THEN
							_Abort := TRUE;
							uiLastBothStep := 0;
							uiResumeStep := 30000;
							uiAbortingStep := 0;
							BoxReady_1st:=FALSE;
						END_IF
						/////////////////////////////////////
				3000:
					
					IF Area= E_RobotArea.InOutConveyor AND Address_B=3 THEN
						uiBothStep:=3100;// Need to control feedout conveyor 
					ELSE
						uiBothStep:=9000;	
					END_IF
				3100:	
					tonDelay.IN := FALSE;
					LowerConveyor.M_MoveBackward();
					IF (NOT FirstSensorOfLowerConveyor) AND (NOT SecondSensorOfLowerConveyor) THEN
						bTimeOutIN:=FALSE;
						uiBothStep:=3200;
					END_IF
					bTimeOutIN:=TRUE;
					//Edited by Jidien Kachu in 2025/10/14
					IF tonTimeOut.Q=TRUE OR Robot._DI1.Error THEN
						strStatus :='FB_RobotAbsMove_V2 Step 30000: Empty Robot timeout';
//						_Error:=TRUE;
						_Abort := TRUE;
						uiLastBothStep := 3000;
						uiResumeStep := 30000;
						uiAbortingStep := 0;
					END_IF	
					///////////////////////////////////////////					
				3200:
					tonDelay.IN := TRUE;
					IF tonDelay.Q THEN
						LowerConveyor.M_MotorStop();
						uiBothStep:=3300;
					END_IF	
					
				
				3300:
					bTimeOutIN:=TRUE;
					tonDelay.IN := FALSE;
					IF 	LowerConveyor.InStopped THEN
						bTimeOutIN:=FALSE;
						BoxReady_2nd:=TRUE;
						uiBothStep:=9999;
					END_IF
					
					//Edited by Jidien Kachu in 2025/10/14
					IF tonTimeOut.Q=TRUE OR Robot._DI1.Error THEN
						strStatus :='FB_RobotAbsMove_V2 Step 30000: Stop Robot timeout';
//						_Error:=TRUE;
						_Abort := TRUE;
						uiLastBothStep := 3200;
						uiResumeStep := 30000;
						uiAbortingStep := 0;
					END_IF	
					///////////////////////////////////////////					
				9000:
						// 檢查 A爪去夾爪時，要確保上層輸送帶是完成的。
						IF Area= E_RobotArea.InOutConveyor AND Address_B = 1 THEN
							IF bCheckUpperCV_ServiceDone THEN
								BoxReady_2nd	 := TRUE;
								_BClampDoingWork := TRUE;
								uiBothStep:=9999;
							END_IF
						ELSE
						BoxReady_2nd	 := TRUE;
						_BClampDoingWork := TRUE;
						uiBothStep:=9999;
						END_IF
				
				9999: //Wait		
				//Edited by Jidien Kachu in 2025/10/14
						IF Robot._DI1.Error THEN
							_Abort := TRUE;
							uiLastBothStep := 3100;
							uiResumeStep := 30000;
							uiAbortingStep := 0;
							BoxReady_2nd:=FALSE;
						END_IF
						/////////////////////////////////////
			// wait reset
			END_CASE
//		END_IF
		
		  

       	  // Robot Abs move
           		 Robot.M_StartRobotAbsMove( GetBox:=Get,
											UseClampA:=UseA,
											UseClampB:=UseB,
											Area:=Area,
											ClampA_Address:=Address_A,
											ClampB_Address:=Address_B,
											BoxReady_1:=BoxReady_1st,
											BoxReady_2:=BoxReady_2nd);	
			IF Get THEN								
				IF _AClampDoingWork AND  NOT Robot._DI1.ClampA_Open THEN
					AClampMoveDone := TRUE;
				END_IF
				IF _BClampDoingWork AND NOT Robot._DI1.ClampB_Open THEN 
					BClampMoveDone := TRUE;
				END_IF
			ELSE
				IF _AClampDoingWork AND Robot._DI1.ClampA_Open THEN
					AClampMoveDone := TRUE;
				END_IF
				IF _BClampDoingWork AND Robot._DI1.ClampB_Open THEN 
					BClampMoveDone := TRUE;
				END_IF
			END_IF
		
		
        IF Robot._DI1.Done THEN
            uiExecutingStep := 30080;
        END_IF
		IF tonRobotTimeOut.Q THEN
			_Abort 		 := TRUE;
			uiResumeStep := 30000;
			strStatus 	 := 'FB_RobotAbsMove_V2 Step 30000: Robot Move timeout';	
		END_IF
		IF Robot._DI1.Error THEN
			_Abort		:= TRUE;
			uiResumeStep:= 30000;
			strStatus	:= CONCAT(STR1 := 'FB_RobotAbsMove_V2 Step 30000:',
								  STR2 := Robot.ErrMsg);
        END_IF
		
    30080: // Check robot command is clear
        
        Robot.M_ResetRobotAbsMove(UseA,UseB);

        IF NOT Robot._DI1.Done THEN
			bTimeOutIN:=FALSE;
			IF Get THEN
				uiExecutingStep := 99000;
			ELSE
				uiExecutingStep := 40000; // go to place step
			END_IF
            
        END_IF    
   		//bTimeOutIN:=TRUE;
		IF tonTimeOut.Q=TRUE THEN
			strStatus := 'FB_RobotAbsMove_V2 Step 30000: Stop Robot timeout';
			_Error:=TRUE;
		END_IF

	40000: // Recheck lowerconveyor Sensor not have box ## Edit by Min 20250416
			
			IF  FirstSensorOfLowerConveyor OR SecondSensorOfLowerConveyor THEN
				bTimeOutIN:=FALSE;
				LowerConveyor.M_MoveBackward();
				uiExecutingStep:=40100;
			ELSE
				uiExecutingStep:=99000;
			END_IF
			bTimeOutIN:=TRUE;
			IF tonTimeOut.Q=TRUE THEN
				strStatus := 'FB_RobotAbsMove_V2 Step 40000: Lowerconveyor Reverse timeout';
				//Edited by Jidien Kachu in 2025/10/14
//				_Error:=TRUE;
				_Abort := TRUE;
				uiResumeStep := 40000;
				uiAbortingStep := 0;
				//////////////////////////////////////
			END_IF	
			
	40100:
			IF NOT (FirstSensorOfLowerConveyor) AND (NOT SecondSensorOfLowerConveyor) THEN
				bTimeOutIN:=FALSE;
				LowerConveyor.M_MotorStop();
				IF LowerConveyor.InStopped THEN
				uiExecutingStep:=99000;
				END_IF
			END_IF
			bTimeOutIN:=TRUE;
			IF tonTimeOut.Q=TRUE THEN
				strStatus :='FB_RobotAbsMove_V2 Step 40100: Lowerconveyor Reverse Stop timeout';
				//Edited by Jidien Kachu in 2025/10/14
//				_Error:=TRUE;
				_Abort := TRUE;
				uiResumeStep := 40100;
				uiAbortingStep := 0;
				//////////////////////////////////////
			END_IF
   
    99000: // process done
        Status    := 'FB_RobotAbsMove_V2 Step 99000: Process completed';
		Cylinder.List.fbLowCV_Block1.M_Retract();
		Cylinder.List.fbLowCV_Press4.M_Retract();
		IF Cylinder.List.fbLowCV_Block1.InRearPosition AND 
			Cylinder.List.fbLowCV_Press4.InRearPosition THEN
			_Executed := TRUE;
			uiBothStep := 0;
			uiSingleClampStep := 0;
		END_IF
END_CASE
IF _Executed THEN
    eState := STATE_DONE;
	uiLastBothStep := 0; //Edited by Jidien Kachu in 2025/10/14
	uiLastSingleClampStep := 0; //Edited by Jidien Kachu in 2025/10/1
ELSIF _Error THEN
	//(iErrorID := ErrorID,UinqueErrorCode=>_UniqueErrorCode);
    eState := STATE_ERROR;
ELSIF NOT Execute THEN
    eState := STATE_RESETTING;
END_IF
IF _Abort OR Abort THEN
	//FUN_UniqueErrorCodeGenerator(iErrorID := ErrorID,UinqueErrorCode=>_UniqueErrorCode);
	eSTATE:=STATE_ABORTING;
END_IF
END_METHOD

METHOD  M_STATE_RESETTING
VAR_INPUT
END_VAR
// Done := false 更改到Dormant 清除確保，上位檢查到done 後可以直接下Execute

CASE uiResettingStep OF

	0:
		bTimeOutIN:=FALSE;
		tonDelay.IN := FALSE	;
		Robot.M_ResetAllCommand();
		Robot.M_ResetRobotAbsMove(TRUE,TRUE);
		uiResettingStep:=100;
		AClampMoveDone	:= FALSE;
		BClampMoveDone	:= FALSE;
		_AClampDoingWork	:= FALSE;
		_BClampDoingWork	:= FALSE;

	100:

		LowerConveyor.M_MotorStop();
		uiResettingStep:=9999;
	9999:
//		Done := FALSE;
//		Busy := FALSE;
		_ResetCompleted:=TRUE;
END_CASE
IF _ResetCompleted THEN
	eSTATE:=STATE_DORMANT;
END_IF
END_METHOD

END_FUNCTION_BLOCK

// ---- Library/20_MachineUnits/21_StorageArea/Service_Robot/FB_WareHouseWithRobotMove_V3.TcPOU
FUNCTION_BLOCK FB_WareHouseWithRobotMove_V3 EXTENDS FB_ObjectBase_V2 IMPLEMENTS IBasicElement
VAR_INPUT
    Robot     : REFERENCE TO FB_FanucRobot_Basic_V2;
    WareHouse : REFERENCE TO FB_WareHouse;
   // Command   : ST_WareHouseWithRobotMove_Command;
    Info	  : st_AutoSixAxisWarehouseParameter;
	Stop	  : BOOL;
	//Edited by Jidien Kachu in 2025/09/25
	iSetRetryCnt	: UINT := 4;
	WarehouseStatus : REFERENCE TO ST_WheelhouseInput; // The warehouse motor and sensor status
END_VAR
VAR_OUTPUT
	AClampMoveDone	: BOOL;
	BClampMoveDone	: BOOL;
  // Status : ST_WareHouseWithRobotMove_Status;
END_VAR
VAR
//	_Abort		: BOOL;
	strStatus	: STRING;
	uiResumeStep : UINT;
	ClampA_WareHouseCoordinates : ST_WareHouseCoordinates;
    ClampB_WareHouseCoordinates : ST_WareHouseCoordinates;
	UseA 	: BOOL;
	UseB	: BOOL;
	TargetWarehouse : E_WareHouse;
	Get 	:BOOL;
	tonTimeout		:TON;
	bTimeOutIN			   : BOOL;
	tonRobotTimeout		:TON;
	bRobotTimeoutIN			   : BOOL;
	_UniqueErrorCode :STRING;
	PreviousStrStatus : STRING;
	PreviousErrorCode : STRING;
	//Edited by Jidien Kachu in 2025/09/25
	iActRetryCnt	: UINT;
	uiBothStep : UINT;
	uiLastBothStep : UINT;
	bRetry: BOOL;
	rtrig: R_TRIG;
	iErrcnt:INT;
	
	_AClampDoingWork	: BOOL;
	_BClampDoingWork	: BOOL;
END_VAR

SUPER^.A10_StateControl();
A00_BasicUnits();

(*============================================================
Create Date : 2025/11/22
Last Update	: 2025/11/22
Change Log  : import Version from TH_Mirror DAS  // Owner : Gamin
============================================================*)

ACTION A00_BasicUnits:
tonTimeOut(IN:= bTimeOutIN AND NOT THIS^.Stop, PT:=T#30S);
tonRobotTimeout(IN:= bRobotTimeoutIN AND NOT THIS^.Stop,PT:=T#60S);
ErrorID :=2400;
rtrig(CLK:= Error);
IF rtrig.Q THEN
	iErrcnt := iErrcnt + 1;
END_IF
END_ACTION

METHOD M_CheckCommand : BOOL // True : Command is useful
VAR_INPUT
END_VAR
VAR
	
END_VAR
// Check command paremeter is correct

IF NOT Info.Warehouse_A AND NOT Info.Warehouse_B THEN
	strStatus:='FB_WareHouseWithRobotMove_V3: Wrong command , No warehouse selected';
	M_CheckCommand:=FALSE;
	RETURN;
ELSIF  Info.Warehouse_A AND  Info.Warehouse_B THEN
	strStatus:='FB_WareHouseWithRobotMove_V3: Wrong command , Both warehouses selected';
	M_CheckCommand:=FALSE;
	RETURN;
ELSIF	Info.Warehouse_A THEN
	TargetWarehouse:=E_WareHouse.WareHouseA;
ELSIF	Info.Warehouse_B THEN
	TargetWarehouse:=E_WareHouse.WareHouseB;
END_IF

IF Info.Get_A <> Info.Get_B THEN
	strStatus:='FB_WareHouseWithRobotMove_V3: Wrong command ,GetA not match to GetB';
	M_CheckCommand:=FALSE;
	RETURN;
	ELSE
		
	Get :=Info.Get_A;
END_IF


CASE LREAL_TO_INT(Info.Layer_A) OF

1,2,3,4,5,6,7,8,9,10:
	//Normal
	// Layer A in correct range
	IF ((Info.Slide_A < 1) OR (Info.Slide_A > 20)) THEN
		strStatus := 'FB_WareHouseWithRobotMove_V3: Command error : Clamp A target slide out of range';
		M_CheckCommand:=FALSE;
		RETURN;
	ELSE
		ClampA_WareHouseCoordinates.Layer:=LREAL_TO_INT(Info.Layer_A);
		ClampA_WareHouseCoordinates.Slide:=LREAL_TO_INT(Info.Slide_A);
   
		UseA:=TRUE;	
	END_IF
	
99:
	UseA:=FALSE;
ELSE
	 strStatus := 'FB_WareHouseWithRobotMove_V3: Command error : Clamp A target layer out of range.';
	 M_CheckCommand:=FALSE;
	 RETURN;
END_CASE


CASE LREAL_TO_INT(Info.Layer_B) OF

1,2,3,4,5,6,7,8,9,10:
//Normal
	// Layer A in correct range
	IF ((Info.Slide_B < 1) OR (Info.Slide_B > 20)) THEN
		strStatus := 'FB_WareHouseWithRobotMove_V3: Command error : Clamp B target slide out of range';
		M_CheckCommand:=FALSE;
		RETURN;
	ELSE
		ClampB_WareHouseCoordinates.Layer:=LREAL_TO_INT(Info.Layer_B);
		ClampB_WareHouseCoordinates.Slide:=LREAL_TO_INT(Info.Slide_B);
		UseB:=TRUE;	
	END_IF
	
99:
		UseB:=FALSE;
ELSE
	 strStatus := 'FB_WareHouseWithRobotMove_V3: Command error : Clamp B target layer out of range.';
	 M_CheckCommand:=FALSE;
	 RETURN;
END_CASE


M_CheckCommand:=TRUE;
END_METHOD

METHOD M_CheckUnitsNotBusy : BOOL
VAR_INPUT
END_VAR
M_CheckUnitsNotBusy := true;
END_METHOD

METHOD M_CheckUnitsReady : BOOL
VAR_INPUT
END_VAR
M_CheckUnitsReady := true;
END_METHOD

METHOD  M_STATE_ABORTED
VAR_INPUT
END_VAR


IF NOT bRetry THEN
	ERROR :=TRUE;
	Busy    := FALSE;
	Aborted := TRUE;
	Status := strStatus;
	UniqueErrorCode:=_UniqueErrorCode;
	_AbortCompleted:=FALSE;
	uiAbortingStep := 0;
END_IF

IF NOT Execute THEN
	eSTATE:=STATE_RESETTING;
END_IF

IF Reset THEN
	bRetry := TRUE;
	ERROR :=FALSE;
	Aborted := FALSE;
END_IF

IF Execute AND bRetry AND NOT Robot.Error AND NOT Robot.Halt THEN

	PreviousStrStatus := strStatus;
	PreviousErrorCode := _UniqueErrorCode;
	uiExecutingStep :=uiResumeStep;
	IF GVL_ADS.MachineState <>E_MachineState.Error THEN
		eSTATE:=STATE_EXECUTING;
	END_IF
	
	iActRetryCnt := iActRetryCnt + 1; //Edited by Jidien Kachu in 2025/09/25
	
	uiBothStep := uiLastBothStep;
END_IF
END_METHOD

METHOD  M_STATE_ABORTING
VAR_INPUT
END_VAR
CASE uiAbortingStep OF
	0 :
			bRetry := FALSE;
			bTimeOutIN:=FALSE;
			bRobotTimeoutIN :=FALSE;
			IF strStatus = PreviousStrStatus THEN
				_UniqueErrorCode :=PreviousErrorCode;
			END_IF
			_Abort :=FALSE;
			(*=====Edited by Jidien Kachu in 2025/09/25=====*)
			Robot.M_ResetAllCommand();
			WareHouse.M_ResetReloadBox();
			WareHouse.M_ResetFeedInBox();
			bRetry := FALSE;
			(*==============================================*)
			
			uiAbortingStep	:= 70;

	70:
			IF Robot._DI1.Error THEN
				uiAbortingStep := 100;
			ELSE
				uiAbortingStep := 9999;
			END_IF
	100:		
			 IF DAS_CoreSys.MachineControl.M_RobotResetCmd() THEN
				 uiAbortingStep := 200;
			 END_IF
	200:
			IF DAS_CoreSys.MachineControl.M_RobotStartCmd() THEN
				 uiAbortingStep := 300;
			 END_IF 
	300:
			IF Robot._DI1.Error THEN
		 		uiAbortingStep := 100;
			ELSE
				uiAbortingStep := 9999;
			END_IF
	9999:	
			_AbortCompleted:=TRUE;
END_CASE

IF _AbortCompleted THEN	
	eSTATE :=STATE_ABORTED;
END_IF
END_METHOD

METHOD  M_STATE_DONE
VAR_INPUT
END_VAR
Busy   := FALSE;
_Error := Error := FALSE;
_Abort := Abort := FALSE;
Done   := TRUE;

IF NOT Execute THEN
    eState := STATE_RESETTING;
END_IF
END_METHOD

METHOD  M_STATE_DORMANT
VAR_INPUT
END_VAR
// Clear FB output
Busy            := FALSE;
Done            := FALSE;
Aborted         := FALSE;
Error           := FALSE;
ErrorID         := 0;
Status          := '';
_ResetCompleted := FALSE;
_Error          := FALSE;
_Executed       := FALSE;
strStatus :='FB_WareHouseWithRobotMove_V3: No Error';
bTimeOutIN :=FALSE;
bRobotTimeoutIN :=FALSE;
uiExecutingStep :=uiResettingStep :=uiResumeStep :=0;
PreviousStrStatus			 :='';
PreviousErrorCode			 :='';
AClampMoveDone	:= FALSE;
BClampMoveDone	:= FALSE;
_AClampDoingWork	:= FALSE;
_BClampDoingWork	:= FALSE;
// Wait Execute command
IF Execute AND NOT Stop  THEN
    eState := STATE_EXECUTING;
END_IF
END_METHOD

METHOD  M_STATE_ERROR
VAR_INPUT
END_VAR
ERROR   :=TRUE;
Busy	:=FALSE;
Status := strStatus;
UniqueErrorCode:=_UniqueErrorCode;
IF NOT Execute THEN	
eSTATE:=STATE_RESETTING;
END_IF
END_METHOD

METHOD  M_STATE_EXECUTING
VAR_INPUT
END_VAR
VAR_INST
	BoxReady_1st : BOOL;
	BoxReady_2nd : BOOL;  
    
    ClampA_WareHouseCoordinates : ST_WareHouseCoordinates;
    ClampB_WareHouseCoordinates : ST_WareHouseCoordinates;
	

	
END_VAR
VAR
	SensorStatus	: BOOL;
END_VAR
// Set Busy active edit by johnson
Busy := TRUE;
(*IF THIS^.Stop THEN // Pending the timeout when Stop signal occur
	bTimeOutIN :=FALSE;
	bRobotTimeoutIN :=FALSE;
END_IF*)
// Service Process
CASE uiExecutingStep OF
	0:
        // Clear variable
       
        bTimeOutIN :=FALSE;
//        uiBothStep := 0;
		uiLastBothStep := 0; //Edited by Jidien Kachu in 2025/10/09
		BoxReady_1st := 0;
		BoxReady_2nd := 0;
        // Check command
        IF M_CheckCommand() THEN
            uiExecutingStep := 10;
		ELSE
			_Error:=TRUE;
        END_IF
		iActRetryCnt := 0; //Edited by Jidien Kachu in 2025/09/25
    10:
        // Start process, check units first
        IF M_CheckUnitsReady() THEN
            uiExecutingStep := 20;
        END_IF
    20:
        // CHeck units not busy state
        IF M_CheckUnitsNotBusy() THEN
            uiExecutingStep := 1000;
        END_IF
   
	1000:   
			// Read  Warehouse coordinate
			ClampA_WareHouseCoordinates := THIS^.ClampA_WareHouseCoordinates;
            ClampB_WareHouseCoordinates := THIS^.ClampB_WareHouseCoordinates;     
			IF UseA AND NOT UseB THEN
				//Only clampA
				uiExecutingStep := 10000;
			ELSIF NOT UseA AND UseB THEN
				//Only ClampB 
				uiExecutingStep := 20000;
			ELSIF UseA AND UseB THEN
				//Both Clamps
				uiExecutingStep := 30000;		
			END_IF
      
	10000:
			IF Get THEN
				IF NOT Robot._DI1.ClampA_Sensor AND Robot._DI1.ClampA_Open THEN		// AClamp has box
					uiExecutingStep := 11000;
				ELSE
					_Abort 	  := TRUE;
					strStatus := 'FB_WareHouseWithRobotMove_V3 Step 10000: Robot Get Box ClampA is open ';




				END_IF
			ELSE
				IF  Robot._DI1.ClampA_Sensor AND NOT Robot._DI1.ClampA_Open THEN	// AClamp has box
					uiExecutingStep := 11000;
				ELSE	
					_Abort 	  := TRUE;
					strStatus := 'FB_WareHouseWithRobotMove_V3 Step 10000: Robot Place Box ClampA not open ';




				END_IF
			END_IF
	
    11000: // Only ClampA 
        IF NOT Robot._DI1.Done THEN
            // Read ClampA Warehouse coordinate
            	ClampA_WareHouseCoordinates := THIS^.ClampA_WareHouseCoordinates;
			
				IF Get THEN// Prepare Box
							//Pick Box
							 WareHouse.M_StartReloadBox(WareHouseSelect := TargetWarehouse, WarehouseCoordinates := ClampA_WareHouseCoordinates);
			
							 // Check Box reload completed
							 IF WareHouse.bReloadBox_Completed THEN
								BoxReady_1st := TRUE;
								_AClampDoingWork := TRUE; // AClamp work edit Gamin 2025/11/21	
							 END_IF
							  // Robot Warehouse move
							 Robot.M_StartWareHousePickUpBox_ClampA(WareHouseSelect := TargetWarehouse,
															   Info            := ClampA_WareHouseCoordinates,
															   BoxReady_1st    := BoxReady_1st);
						// make sure robot doing AClamp done
						IF _AClampDoingWork AND  NOT Robot._DI1.ClampA_Open THEN
								AClampMoveDone := TRUE;
						END_IF
					  	
				ELSE
						//Place Box
							WareHouse.M_StartFeedInBox(WareHouseSelect := TargetWarehouse, WarehouseCoordinates := ClampA_WareHouseCoordinates);
		
							 // Check Box reload completed
							 IF WareHouse.bFeedInBox_Completed THEN
								 BoxReady_1st := TRUE;
								 _AClampDoingWork := TRUE; // AClamp work edit Gamin 2025/11/21	
							 END_IF				
									   
							Robot.M_StartWareHousePlaceBox_ClampA(WareHouseSelect 	:= TargetWarehouse,
																	Info            := ClampA_WareHouseCoordinates,
																	BoxReady_1st    := BoxReady_1st);
						IF _AClampDoingWork AND robot._DI1.ClampA_Open THEN 
							AClampMoveDone := TRUE;
						END_IF
			   END_IF
			   
        ELSE
            uiExecutingStep := 12000;
        END_IF
		

		bTimeOutIN:=TRUE;
		IF tonTimeout.Q OR Robot.Error THEN
			_Abort := TRUE;
            uiResumeStep := 11000;
			strStatus:='FB_WareHouseWithRobotMove_V3 Step 11000: Robot Move Timeout';




		END_IF
		
    12000:
        Robot.M_ResetAllCommand(); // Clear command and go to place box
		bTimeOutIN :=FALSE;
		bRobotTimeoutIN :=FALSE;
		
        IF NOT Robot._DI1.Done THEN
            uiExecutingStep := 99000; 
        END_IF
    
   20000:
   			IF Get THEN
				IF NOT Robot._DI1.ClampB_Sensor AND Robot._DI1.ClampB_Open THEN	// BClamp has box
					uiExecutingStep := 21000;
				ELSE
					_Abort	:= TRUE;
					strStatus := 'FB_WareHouseWithRobotMove_V3 Step 20000: Robot Get Box ClampB is open ';




				END_IF
			ELSE
				IF Robot._DI1.ClampB_Sensor AND NOT Robot._DI1.ClampB_Open THEN	// BClamp has box
					uiExecutingStep := 21000;
				ELSE
					_Abort	:= TRUE;
					strStatus := 'FB_WareHouseWithRobotMove_V3 Step 20000: Robot Place Box ClampB not open ';




				END_IF
			END_IF
	
   21000: // Only ClampB
        IF NOT Robot._DI1.Done THEN
            			
			IF Get THEN// Prepare Box
				//Pick Box
				 WareHouse.M_StartReloadBox(WareHouseSelect := TargetWarehouse, WarehouseCoordinates := ClampB_WareHouseCoordinates);

				 // Check Box reload completed
				 IF WareHouse.bReloadBox_Completed THEN
					 BoxReady_2nd := TRUE;
					 _BClampDoingWork := TRUE;	// BClamp work edit Gamin 2025/11/21	
				 END_IF
				  // Robot Warehouse move
				 Robot.M_StartWareHousePickUpBox_ClampB(WareHouseSelect := TargetWarehouse,
												   Info            := ClampB_WareHouseCoordinates,
												   BoxReady_2nd    := BoxReady_2nd);
				IF _BClampDoingWork AND NOT Robot._DI1.ClampB_Open THEN 
					BClampMoveDone := TRUE;
				END_IF
			ELSE
				//Place Box
				WareHouse.M_StartFeedInBox(WareHouseSelect := TargetWarehouse, WarehouseCoordinates := ClampB_WareHouseCoordinates);

				 // Check Box reload completed
				 IF WareHouse.bFeedInBox_Completed THEN
					 BoxReady_2nd := TRUE;
					 _BClampDoingWork := TRUE;	// BClamp work edit Gamin 2025/11/21	
				 END_IF				
						   
				Robot.M_StartWareHousePlaceBox_ClampB (WareHouseSelect := TargetWarehouse,
											   Info            := ClampB_WareHouseCoordinates,
											   BoxReady_2nd    := BoxReady_2nd);
				IF _BClampDoingWork AND Robot._DI1.ClampB_Open THEN 
					BClampMoveDone := TRUE;
				END_IF
           END_IF
        ELSE
            uiExecutingStep := 22000;
        END_IF
		

		bTimeOutIN:=TRUE;
		IF tonTimeout.Q OR Robot.Error THEN
			_Abort := TRUE;
            uiResumeStep := 21000;
			strStatus:='FB_WareHouseWithRobotMove_V3 Step 21000: Robot Move Timeout';




		END_IF
		
    22000:
        Robot.M_ResetAllCommand(); // Clear command and go to place box
		bTimeOutIN :=FALSE;
		bRobotTimeoutIN :=FALSE;
		
        IF NOT Robot._DI1.Done THEN
            uiExecutingStep := 99000; 
        END_IF
		
	30000:
			IF Get THEN
				IF  NOT Robot._DI1.ClampA_Sensor AND Robot._DI1.ClampA_Open AND 
					NOT Robot._DI1.ClampB_Sensor AND Robot._DI1.ClampB_Open THEN
					uiExecutingStep := 31000;
				ELSE
					_Abort	:= TRUE;
					strStatus := 'FB_WareHouseWithRobotMove_V3 Step 30000: Robot both Clamp Get Box ,  Clamp not open';




				END_IF
			ELSE
				IF  Robot._DI1.ClampA_Sensor AND NOT Robot._DI1.ClampA_Open AND 
				 	Robot._DI1.ClampB_Sensor AND NOT Robot._DI1.ClampB_Open THEN
					uiExecutingStep := 31000;
				ELSE
					_Abort	:= TRUE;
					strStatus := 'FB_WareHouseWithRobotMove_V3 Step 30000: Robot both Clamp Place Box , Clamp has open';




				END_IF 
			END_IF
				
    31000: // Both Clampss
        		
		IF Get THEN //BOth clamps pick
			
				CASE uiBothStep OF
					0: // ClampA target slide move the box to front side
						WareHouse.M_StartReloadBox(WareHouseSelect      := TargetWarehouse,
												   WarehouseCoordinates := ClampA_WareHouseCoordinates);
						bTimeOutIN :=TRUE;
						IF tonTimeout.Q THEN
							_Abort := TRUE;
							uiAbortingStep := 0;
							uiLastBothStep := 0;
							uiResumeStep := 31000;
							(*==============================================*)
							strStatus:='FB_WareHouseWithRobotMove_V3 Step 31000: Clamp A reload timeout';




						END_IF
					   
						IF WareHouse.bReloadBox_Completed THEN
							bTimeOutIN :=FALSE;
							BoxReady_1st     := TRUE;
							_AClampDoingWork := TRUE;	//AClamp work edit Gamin 2025/11/21	
							uiBothStep := 10;
						END_IF
		
					10: // wait Robot Allow continue
							WareHouse.M_ResetReloadBox();
						IF Robot._DI1.Notification  THEN // AND
							IF NOT WareHouse.bReloadBox_Completed THEN					
								uiBothStep := 15;
							END_IF
						END_IF
	
						IF Robot._DI1.Error THEN
							_Abort := TRUE;
							BoxReady_1st := FALSE;
							_AClampDoingWork := FALSE;
							uiAbortingStep := 0;
							uiLastBothStep := 0;
							uiResumeStep := 31000;
							strStatus:='FB_WareHouseWithRobotMove_V3 Step 31000: Robot Has Fault';




						END_IF

					15:	IF NOT WareHouse._stWarehouseList.ASide_Layers[ClampA_WareHouseCoordinates.Layer].stStatus.bSlides[ClampA_WareHouseCoordinates.Slide] THEN
							 uiBothStep := 17;	
						 END_IF
					17:
						IF info.Warehouse_A THEN 
							SensorStatus := NOT WarehouseStatus.WheelhouseA.arLayer[ClampA_WareHouseCoordinates.Layer].Line[ClampA_WareHouseCoordinates.Slide];
							IF SensorStatus THEN
								uiBothStep := 20;
							END_IF
						ELSIF info.Warehouse_B THEN
							SensorStatus := NOT WarehouseStatus.WheelhouseB.arLayer[ClampA_WareHouseCoordinates.Layer].Line[ClampA_WareHouseCoordinates.Slide];
							IF SensorStatus THEN
								uiBothStep := 20;
							END_IF
						END_IF
						 
					20: // ClampB target slide move the box to front slide
						WareHouse.M_StartReloadBox(WareHouseSelect := TargetWarehouse, WarehouseCoordinates := ClampB_WareHouseCoordinates);
						bTimeOutIN :=TRUE;
						IF WareHouse.bReloadBox_Completed THEN
							bTimeOutIN :=FALSE;
							BoxReady_2nd     := TRUE;
							_BClampDoingWork := TRUE;
							uiBothStep := 99;
						END_IF
						IF tonTimeout.Q THEN
								_Abort := TRUE;
								uiAbortingStep := 0;
								uiLastBothStep := 20;
								BoxReady_2nd     := FALSE;
								_BClampDoingWork := FALSE;
								uiResumeStep := 31000;
							(*==============================================*)
							strStatus:='FB_WareHouseWithRobotMove_V3 Step 31000: Clamp B reload timeout';




						END_IF
					99:
						WareHouse.M_ResetReloadBox();
				// wait reset
				END_CASE	
	
				Robot.M_StartWareHousePickUpBox_ClampBoth(WareHouseSelect := TargetWarehouse,
														  ClampA_Info     := ClampA_WareHouseCoordinates,
														  ClampB_Info     := ClampB_WareHouseCoordinates,
														  BoxReady_1st    := BoxReady_1st,
														  BoxReady_2nd    := BoxReady_2nd);
													  
				bRobotTimeoutIN :=TRUE;
				IF Robot.Error OR tonRobotTimeout.Q THEN
					_Abort := TRUE;
					uiAbortingStep := 0;
					IF NOT BoxReady_1st THEN
						BoxReady_1st     := FALSE;
						_AClampDoingWork := FALSE;
						uiLastBothStep := 0;
						uiResumeStep := 31000;
					ELSE
						uiLastBothStep := 20;
						BoxReady_2nd     := FALSE;
						_BClampDoingWork := FALSE;
						uiResumeStep := 31000;
					END_IF
					(*==============================================*)
					strStatus:='FB_WareHouseWithRobotMove_V3 Step 31000: Robot Has Fault';




				END_IF
			
			IF _AClampDoingWork AND NOT Robot._DI1.ClampA_Open THEN
				AClampMoveDone := TRUE;
			END_IF
			IF _BClampDoingWork AND NOT Robot._DI1.ClampB_Open THEN
				BClampMoveDone := TRUE;
			END_IF
		ELSE
				 
					CASE uiBothStep OF
					  
					   0: // ClampA target slide move the box to front side
						WareHouse.M_StartFeedInBox(WareHouseSelect      := TargetWarehouse,
												   WarehouseCoordinates := ClampA_WareHouseCoordinates);
		
					   bTimeOutIN :=TRUE;
						IF WareHouse.bFeedInBox_Completed THEN
							bTimeOutIN :=FALSE;
							BoxReady_1st     := TRUE;
							_AClampDoingWork := TRUE;
							uiBothStep := 10;
						END_IF
						IF tonTimeout.Q THEN
							(*=====Edited by Jidien Kachu in 2025/09/25=====*)

								_Abort := TRUE;
								uiAbortingStep := 0;
								uiResumeStep := 31000;
								BoxReady_1st     := FALSE;
								_AClampDoingWork := FALSE;

							(*==============================================*)
							strStatus:='FB_WareHouseWithRobotMove_V3 Step 31000: Clamp A Feedin timeout';




						END_IF
		
					10: // wait Robot Allow continue
							WareHouse.M_ResetFeedInBox();
						 IF Robot._DI1.Notification THEN //AND
							IF NOT WareHouse.bFeedInBox_Completed THEN
								
								uiBothStep := 15;
							END_IF
						END_IF
						(*=====Edited by Jidien Kachu in 2025/10/27=====*)
						IF Robot._DI1.Error THEN
							_Abort := TRUE;
							uiAbortingStep := 0;
							uiLastBothStep := 0;
							uiResumeStep := 31000;
							BoxReady_1st     := FALSE;
							_AClampDoingWork := FALSE;
							strStatus:='FB_WareHouseWithRobotMove_V3 Step 31000: Robot Has Fault';




						END_IF
						(*==============================================*)
					15:  
						uiBothStep := 20;
					
					20: // ClampB target slide move the box to front slide
						WareHouse.M_StartFeedInBox(WareHouseSelect := TargetWarehouse, WarehouseCoordinates := ClampB_WareHouseCoordinates);
						bTimeOutIN :=TRUE;
						IF WareHouse.bFeedInBox_Completed THEN
							bTimeOutIN :=FALSE;
							BoxReady_2nd     := TRUE;
							_BClampDoingWork := TRUE;
							uiBothStep := 99;
						END_IF
						IF tonTimeout.Q THEN
							(*=====Edited by Jidien Kachu in 2025/09/25=====*)
								_Abort := TRUE;
								uiAbortingStep := 0;
								uiLastBothStep := 20;
								BoxReady_2nd 	 := FALSE;
								_BClampDoingWork := FALSE;
							(*==============================================*)
							strStatus:='FB_WareHouseWithRobotMove_V3 Step 31000: Clamp B Feedin timeout';




						END_IF
					99: 
						WareHouse.M_ResetFeedInBox();
		
				END_CASE

       		 Robot.M_StartWareHousePlaceUpBox_ClampBoth(WareHouseSelect := TargetWarehouse,
                                                  ClampA_Info     := ClampA_WareHouseCoordinates,
                                                  ClampB_Info     := ClampB_WareHouseCoordinates,
                                                  BoxReady_1st    := BoxReady_1st,
                                                  BoxReady_2nd    := BoxReady_2nd);
												  
				bRobotTimeoutIN :=TRUE;
			(*=====Edited by Jidien Kachu in 2025/09/25=====*)
				IF Robot.Error OR tonRobotTimeout.Q THEN
					_Abort := TRUE;
					uiAbortingStep := 0;
					IF NOT BoxReady_1st THEN
						uiLastBothStep := 0;
						uiResumeStep := 31000;
						BoxReady_1st := FALSE;
						_AClampDoingWork := FALSE;
					ELSE
						uiResumeStep := 31000;
						uiLastBothStep := 20;
						BoxReady_2nd := FALSE;
						_BClampDoingWork := FALSE;
					END_IF
					strStatus:='FB_WareHouseWithRobotMove_V3 Step 31000: Robot Has Fault';




				END_IF
			IF _AClampDoingWork AND  Robot._DI1.ClampA_Open THEN
				AClampMoveDone := TRUE;
			END_IF
			IF _BClampDoingWork AND  Robot._DI1.ClampB_Open THEN
				BClampMoveDone := TRUE;
			END_IF
		END_IF
		
        IF Robot._DI1.Done THEN
			uiBothStep := 0;
            uiExecutingStep := 31080;
        END_IF
		
    31080: // Check robot command is clear
		
        WareHouse.M_ResetReloadBox();
        WareHouse.M_ResetFeedInBox();
        Robot.M_ResetAllCommand();
		bTimeOutIN :=FALSE;
		bRobotTimeoutIN :=FALSE;
		
        IF NOT Robot._DI1.Done THEN
            uiExecutingStep := 99000; // go to place step
        END_IF    
   
   
    99000: // process done
                Status    := 'FB_WareHouseWithRobotMove_V3 Step 99000: Process completed';
        _Executed := TRUE;
END_CASE
IF _Executed THEN
    eState := STATE_DONE;
	uiLastBothStep := 0; //Edited by Jidien Kachu in 2025/10/27
	uiBothStep := 0; //Edited by Jidien Kachu in 2025/10/27
ELSIF _Error THEN
    eState := STATE_ERROR;
ELSIF NOT Execute THEN
    eState := STATE_RESETTING;
END_IF
IF _Abort OR Abort THEN
	eSTATE:=STATE_ABORTING;
END_IF
END_METHOD

METHOD  M_STATE_RESETTING
VAR_INPUT
END_VAR
// Done := false 更改到Dormant 清除確保，上位檢查到done 後可以直接下Execute

CASE uiResettingStep OF

	0:
		bTimeOutIN :=FALSE;
		bRobotTimeoutIN :=FALSE;
		Robot.M_ResetAllCommand();
		uiResettingStep:=9999;
		WareHouse.M_ResetFeedInBox();
		WareHouse.M_ResetReloadBox();
		uiLastBothStep := 0; //Edited by Jidien Kachu in 2025/10/27
		uiBothStep := 0; //Edited by Jidien Kachu in 2025/10/27
//		Robot.M_CycleStop(TRUE);
		AClampMoveDone := FALSE;
		BClampMoveDone := FALSE;
		_AClampDoingWork := FALSE;
		_BClampDoingWork := FALSE;

	9999:
//		Robot.M_CycleStop(FALSE);
//		Done := FALSE;
//		Busy := FALSE;
		_ResetCompleted:=TRUE;
END_CASE
IF _ResetCompleted THEN
	eSTATE:=STATE_DORMANT;
END_IF
END_METHOD

END_FUNCTION_BLOCK

// ---- Library/20_MachineUnits/21_StorageArea/Service_Robot/FB_FeedInRoundBeltBoxToWareHouse.TcPOU
(*
	FB_FeedInRoundBeltBoxToWareHouse
	功能：從圓帶取盒子放回倉儲 (與 FB_ReloadRoundBeltBoxWithRobot_V2 反向操作)
	流程：圓帶移動到站位 → 手臂 AbsMove 從圓帶取盒 → 手臂放盒到倉儲
	安全卡控：手臂進入圓帶區域時，取得圓帶控制權，圓帶不可移動
*)
FUNCTION_BLOCK FB_FeedInRoundBeltBoxToWareHouse EXTENDS FB_ObjectBase_V2 IMPLEMENTS IBasicElement
VAR_INPUT
    // ===== 外部元件參考 =====
    Robot         : REFERENCE TO FB_FanucRobot_Basic_V2; // Fanuc 手臂
	RoundBelt	  : REFERENCE TO FB_RoundBeltService;    // 圓帶服務
    WareHouse     : REFERENCE TO FB_WareHouse;           // 倉儲區
	Input         : ST_InputTable;                        // IO 輸入表
    Info          : ST_FeedInToWareHouseBox_Info;         // C# ADS 餵入的動作參數 (A爪/B爪 取盒位置、放盒目標)
    Stop          : BOOL;                                 // 停止訊號，暫停 Timeout 計時

	// ===== Batch handshake mode (opt-in) =====
	// 由 Batch FB 設為 TRUE 啟用 ActionRecord + FeedBack/ReadComplete 握手
	// 預設 FALSE → 走原本流程,完成後直接 _Executed,不產生 ActionRecord (向後相容)
	HandshakeMode : BOOL;
	ReadComplete  : BOOL;	// (HandshakeMode 時) C# 讀取陣列完成確認
END_VAR
VAR_OUTPUT
	AClampMoveDone	: BOOL;  // A爪動作完成旗標，供 C# 寫入 SQL
	BClampMoveDone	: BOOL;  // B爪動作完成旗標，供 C# 寫入 SQL

	// ===== Batch handshake outputs (僅 HandshakeMode=TRUE 時填入) =====
	ActionRecords	: ARRAY[0..39] OF ST_FeedInRBActionRecord;	// 動作紀錄陣列
	ActionIndex		: INT;		// 已記錄筆數 (0..40)
	FeedBack		: BOOL;		// TRUE = 流程完成,陣列可讀取 (PLC → C#)
END_VAR
VAR
    strStatus         : STRING;   // 錯誤/狀態訊息
    tonTimeOut        : TON;      // 通用逾時計時器 (120s),由各 step 自行呼叫 (IN:=TRUE, PT:=)
    tonReadComplete   : TON;      // (HandshakeMode) C# 讀取確認逾時 (15s)
    _UniqueErrorCode  : STRING;
    PreviousStrStatus : STRING;   // Resume 前的狀態訊息
    PreviousErrorCode : STRING;   // Resume 前的錯誤碼
    A2_Sensor         : BOOL;    // 圓帶 A2 位置感測器
    A3_Sensor         : BOOL;    // 圓帶 A3 位置感測器

	// ===== 爪工作旗標 =====
	_AClampDoingWork	: BOOL;  // A爪正在執行
	_BClampDoingWork	: BOOL;  // B爪正在執行

	// ========== Resume 續做機制 ==========
	uiResumeStep	: UDINT := 0;	// 錯誤發生時記錄的步驟，供續做使用

	// =========== Aborted =================
	_bRetry			: BOOL;

	// Step 切換偵測 (timer 乾淨重置,避免 tonTimeOut.IN 殘留 TRUE 造成跨 step 不歸零)
	uiExecutingStep_Last : UDINT;

END_VAR

SUPER^.A10_StateControl();
A00_BasicUnits();
A2_Sensor := Input.bRoundBelt_ChangeZoneA2Detect_Sensor;
A3_Sensor := Input.bRoundBelt_ChangeZoneA3Detect_Sensor;

(*============================================================
Create Date : 2026/03/18
Last Update	: 2026/04/20
Change Log  : 2026/03/18，Initial version - Pick box from RoundBelt and place to WareHouse
			  2026/03/23，修正續做，新增手臂先在aborting清除錯誤，
			  2026/04/14，新的FB新增回拔輸送帶放盒位置支援，ActionRecords功能，把這一隻舊的移除至Old_version_Service 資料夾內。
			  2026/04/20，更新版本，將舊的移至Old Service 資料夾內，修正ActionRecords 未上拋問題。
============================================================*)

ACTION A00_BasicUnits:
// Timer 由各 step 自行呼叫並傳 IN/PT,此處不做 freerun call,
// 避免「IN 殘留 TRUE」造成 step 切換後 timer 不歸零。
END_ACTION

METHOD M_AppendActionRecord_ClampA
VAR_INPUT
END_VAR
IF NOT HandshakeMode OR ActionIndex >= 40 THEN
	RETURN;
END_IF

ActionRecords[ActionIndex].PickStation := UINT_TO_INT(info.ClampA_Setting.RoundBeltSetting.Station);
ActionRecords[ActionIndex].PickCarrier := info.ClampA_Setting.RoundBeltSetting.ReloadCarrier;
ActionRecords[ActionIndex].Clamp := 0;

IF info.ClampA_Setting.PlaceArea = E_FeedInToWareHouse_PlaceArea.WareHouseA
OR info.ClampA_Setting.PlaceArea = E_FeedInToWareHouse_PlaceArea.WareHouseB THEN
	ActionRecords[ActionIndex].DestType := 0;
	IF info.ClampA_Setting.PlaceArea = E_FeedInToWareHouse_PlaceArea.WareHouseA THEN
		ActionRecords[ActionIndex].WareHouse := 1;
	ELSE
		ActionRecords[ActionIndex].WareHouse := 2;
	END_IF
	ActionRecords[ActionIndex].Layer := info.ClampA_Setting.WareHouseSetting.Layer;
	ActionRecords[ActionIndex].Slide := info.ClampA_Setting.WareHouseSetting.Slide;
	ActionRecords[ActionIndex].PullOutSide := 0;
ELSE
	ActionRecords[ActionIndex].DestType := 1;
	ActionRecords[ActionIndex].WareHouse := 0;
	ActionRecords[ActionIndex].Layer := 0;
	ActionRecords[ActionIndex].Slide := 0;
	IF info.ClampA_Setting.PlaceArea = E_FeedInToWareHouse_PlaceArea.PullOutInner THEN
		ActionRecords[ActionIndex].PullOutSide := 0;
	ELSE
		ActionRecords[ActionIndex].PullOutSide := 1;
	END_IF
END_IF

ActionIndex := ActionIndex + 1;
END_METHOD

METHOD M_AppendActionRecord_ClampB
VAR_INPUT
END_VAR
IF NOT HandshakeMode OR ActionIndex >= 40 THEN
	RETURN;
END_IF

ActionRecords[ActionIndex].PickStation := UINT_TO_INT(info.ClampB_Setting.RoundBeltSetting.Station);
ActionRecords[ActionIndex].PickCarrier := info.ClampB_Setting.RoundBeltSetting.ReloadCarrier;
ActionRecords[ActionIndex].Clamp := 1;

IF info.ClampB_Setting.PlaceArea = E_FeedInToWareHouse_PlaceArea.WareHouseA
OR info.ClampB_Setting.PlaceArea = E_FeedInToWareHouse_PlaceArea.WareHouseB THEN
	ActionRecords[ActionIndex].DestType := 0;
	IF info.ClampB_Setting.PlaceArea = E_FeedInToWareHouse_PlaceArea.WareHouseA THEN
		ActionRecords[ActionIndex].WareHouse := 1;
	ELSE
		ActionRecords[ActionIndex].WareHouse := 2;
	END_IF
	ActionRecords[ActionIndex].Layer := info.ClampB_Setting.WareHouseSetting.Layer;
	ActionRecords[ActionIndex].Slide := info.ClampB_Setting.WareHouseSetting.Slide;
	ActionRecords[ActionIndex].PullOutSide := 0;
ELSE
	ActionRecords[ActionIndex].DestType := 1;
	ActionRecords[ActionIndex].WareHouse := 0;
	ActionRecords[ActionIndex].Layer := 0;
	ActionRecords[ActionIndex].Slide := 0;
	IF info.ClampB_Setting.PlaceArea = E_FeedInToWareHouse_PlaceArea.PullOutInner THEN
		ActionRecords[ActionIndex].PullOutSide := 0;
	ELSE
		ActionRecords[ActionIndex].PullOutSide := 1;
	END_IF
END_IF

ActionIndex := ActionIndex + 1;
END_METHOD

METHOD M_CheckCommand : BOOL
VAR_INPUT
END_VAR
VAR_INST
	CheckBehavior : BOOL;
END_VAR
VAR
	I: INT;
END_VAR
// Memory clear
CheckBehavior := FALSE;
// Check command is correct
IF info.ClampA_Setting.Behavior = E_ClampWork.Work OR info.ClampB_Setting.Behavior = E_ClampWork.Work THEN
	CheckBehavior := TRUE;
ELSE
	CheckBehavior := FALSE;
END_IF

M_CheckCommand := CheckBehavior;
END_METHOD

METHOD M_CheckUnitsNotBusy : BOOL
VAR_INPUT
END_VAR
M_CheckUnitsNotBusy := true;
END_METHOD

METHOD M_CheckUnitsReady : BOOL
VAR_INPUT
END_VAR
M_CheckUnitsReady := true;
END_METHOD

(* 根據 A爪/B爪 的 Behavior 和 PlaceArea 判斷動作模式
   - 單爪A/B：從圓帶取盒後放到 WareHouseA 或 WareHouseB
   - 雙爪：兩爪各自從圓帶取盒，放到指定的倉儲 (可同倉或不同倉)
*)
METHOD M_SelectActionMode : E_FeedInToWareHouseAction
VAR_INPUT
END_VAR
// 判斷 A爪/B爪 是否有工作，以及放盒目標倉儲
IF info.ClampA_Setting.Behavior <> E_ClampWork.Work AND info.ClampB_Setting.Behavior <> E_ClampWork.Work THEN
	M_SelectActionMode := E_FeedInToWareHouseAction.Undefined;
ELSIF info.ClampA_Setting.Behavior = E_ClampWork.Work AND info.ClampB_Setting.Behavior <> E_ClampWork.Work THEN
	IF info.ClampA_Setting.PlaceArea = E_FeedInToWareHouse_PlaceArea.WareHouseA THEN
		M_SelectActionMode := E_FeedInToWareHouseAction.ClampA_WareHouseA;
	ELSIF info.ClampA_Setting.PlaceArea = E_FeedInToWareHouse_PlaceArea.WareHouseB THEN
		M_SelectActionMode := E_FeedInToWareHouseAction.ClampA_WareHouseB;
	END_IF
ELSIF info.ClampA_Setting.Behavior <> E_ClampWork.Work AND info.ClampB_Setting.Behavior = E_ClampWork.Work THEN
	IF info.ClampB_Setting.PlaceArea = E_FeedInToWareHouse_PlaceArea.WareHouseA THEN
		M_SelectActionMode := E_FeedInToWareHouseAction.ClampB_WareHouseA;
	ELSIF info.ClampB_Setting.PlaceArea = E_FeedInToWareHouse_PlaceArea.WareHouseB THEN
		M_SelectActionMode := E_FeedInToWareHouseAction.ClampB_WareHouseB;
	END_IF
ELSIF info.ClampA_Setting.Behavior = E_ClampWork.Work AND info.ClampB_Setting.Behavior = E_ClampWork.Work THEN
	IF info.ClampA_Setting.PlaceArea = E_FeedInToWareHouse_PlaceArea.WareHouseA THEN
		IF info.ClampB_Setting.PlaceArea = E_FeedInToWareHouse_PlaceArea.WareHouseA THEN
			M_SelectActionMode := E_FeedInToWareHouseAction.A_WareHouseA_B_WareHouseA;
		ELSIF info.ClampB_Setting.PlaceArea = E_FeedInToWareHouse_PlaceArea.WareHouseB THEN
			M_SelectActionMode := E_FeedInToWareHouseAction.A_WareHouseA_B_WareHouseB;
		END_IF
	ELSIF info.ClampA_Setting.PlaceArea = E_FeedInToWareHouse_PlaceArea.WareHouseB THEN
		IF info.ClampB_Setting.PlaceArea = E_FeedInToWareHouse_PlaceArea.WareHouseA THEN
			M_SelectActionMode := E_FeedInToWareHouseAction.A_WareHouseB_B_WareHouseA;
		ELSIF info.ClampB_Setting.PlaceArea = E_FeedInToWareHouse_PlaceArea.WareHouseB THEN
			M_SelectActionMode := E_FeedInToWareHouseAction.A_WareHouseB_B_WareHouseB;
		END_IF
	END_IF
END_IF
END_METHOD

METHOD  M_STATE_ABORTED
VAR_INPUT
END_VAR
IF NOT _bRetry THEN
	Busy    := FALSE;
	Error	:= TRUE;
	Aborted := TRUE;
	UniqueErrorCode := _UniqueErrorCode;
	uiAbortingStep  := 0;
	_AbortCompleted := FALSE;
	Status := strStatus;
END_IF

IF reset THEN
	_bRetry := TRUE;
	Error	:= FALSE;
	Aborted := FALSE;
	_Abort  := FALSE;
END_IF

// ============================================================
// Resume 續做機制：保持 Execute 並按 Reset 可從錯誤點繼續執行
// ============================================================
IF NOT Execute THEN
	eState := STATE_RESETTING;
ELSIF Execute AND _bRetry AND NOT Robot._DI1.Error AND NOT Robot.Halt THEN
	// Resume 模式：確認 Robot 不在暫停且無錯誤，從儲存的步驟繼續執行
	Status := '';
	uiExecutingStep := uiResumeStep;
	PreviousStrStatus := strStatus;
	PreviousErrorCode := _UniqueErrorCode;
	IF GVL_ADS.MachineState <>E_MachineState.Error THEN
		eSTATE:=STATE_EXECUTING;
	END_IF
END_IF
END_METHOD

METHOD  M_STATE_ABORTING
VAR_INPUT
END_VAR
CASE uiAbortingStep OF
	0:
			_Abort 				:= FALSE;
			_bRetry				:= FALSE;
			tonTimeOut(IN := FALSE);

			// 清除 Robot DO handshake 和周邊狀態（不管 Robot 是 Error 還是 Held）
	
			(* 
				comment edited By Gamin ，
				1. 續做不能清除手臂命令，如果是做雙爪夾盒，A爪做完B爪報錯進入到續做流程，如果在此清除掉手臂命令
					，後續回到executing 動作，此時的情境為A 已做完已夾完盒，等同於給手臂重新做的命令，，會有危險，
				2. 在Service 執行期間進入到錯誤狀態也不能清除圓帶的使用權，以免被其他的Serivce 搶走，會有危險
				3.  A、B done 不能清除，這旗標也可算是代表手臂該爪的動作完成，
				   如果A爪完成，B爪報錯，續做只接續著做B爪，這樣Service 結束就只會有B done。
			*)
//			Robot.M_ResetAllCommand();
//			WareHouse.M_ResetFeedInBox();
//			DAS_CoreSys.MachineControl.fbAllocateArea.M_ResetReloadRoundBeltAction();
//			DAS_CoreSys.MachineControl.fbAllocateArea.M_ReleaseRoundBeltAccess(ControlAccess := E_RoundBeltControlAccess.FanucRobot);
//			AClampMoveDone	 := FALSE;
//			BClampMoveDone	 := FALSE;
//			_AClampDoingWork := FALSE;
//			_BClampDoingWork := FALSE;

			uiAbortingStep := 100;
    100:
			IF Robot._DI1.Error THEN
				uiAbortingStep := 200;
			ELSE
				uiAbortingStep := 9999;
			END_IF
			
	200:		
			 IF DAS_CoreSys.MachineControl.M_RobotResetCmd() THEN
				 uiAbortingStep := 300;
			 END_IF
			 
	300:
			IF DAS_CoreSys.MachineControl.M_RobotStartCmd() THEN
				 uiAbortingStep := 400;
			 END_IF 
			 
	400:
			IF Robot._DI1.Error THEN
		 		uiAbortingStep := 200;
			ELSE
				uiAbortingStep := 9999;
			END_IF
			
	9999:
			_AbortCompleted := TRUE;
END_CASE


IF _AbortCompleted THEN
    eState := STATE_Aborted;
END_IF
END_METHOD

METHOD  M_STATE_DONE
VAR_INPUT
END_VAR
Busy   := FALSE;
_Error := Error := FALSE;
_Abort := Abort := FALSE;
Done   := TRUE;

IF NOT Execute THEN
    eState := STATE_RESETTING;
END_IF
END_METHOD

METHOD  M_STATE_DORMANT
VAR_INPUT
END_VAR
// 清除 FB 所有輸出與內部狀態
Busy            := FALSE;
Done            := FALSE;
Aborted         := FALSE;
Error           := FALSE;
ErrorID         := 0;
Status          := '';
_ResetCompleted := FALSE;
_Error          := FALSE;
_Executed       := FALSE;
_Abort			:= FALSE;

uiExecutingStep := 0;
uiAbortingStep	:= 0;
uiResettingStep := 0;
uiResumeStep    := 0;
uiExecutingStep_Last := 0;

// Timer 完整歸零 (用實際 FB call,不是只設屬性)
tonTimeOut(IN := FALSE);

PreviousStrStatus := '';
PreviousErrorCode := '';
_UniqueErrorCode := '0';

AClampMoveDone 	 := FALSE;
BClampMoveDone 	 := FALSE;
_AClampDoingWork := FALSE;
_BClampDoingWork := FALSE;
_AbortCompleted	 := FALSE;

_bRetry			:= FALSE;

// HandshakeMode: 清 ActionRecord / handshake 旗標
FeedBack := FALSE;
ActionIndex := 0;
MEMSET(ADR(ActionRecords), 0, SIZEOF(ActionRecords));
tonReadComplete(IN := FALSE);

// 等待 Execute 命令啟動
IF Execute AND NOT Stop THEN
    eState := STATE_EXECUTING;
END_IF
END_METHOD

METHOD  M_STATE_ERROR
VAR_INPUT
END_VAR
UniqueErrorCode	:= _UniqueErrorCode;
Error			:= TRUE;
Busy			:= FALSE;
status			:= strStatus;


IF NOT Execute THEN
    eState := STATE_RESETTING;
END_IF
END_METHOD

(*
	M_STATE_EXECUTING 主執行流程
	Step 配置：
	  0~1100    : 初始化、命令檢查、模式選擇
	  10000~10080 : A爪單爪 - 從圓帶取盒
	  20000~20080 : B爪單爪 - 從圓帶取盒
	  30000~31080 : 雙爪 - 從圓帶取盒 (先A後B，支援同站/不同站)
	  60000~61080 : A爪單爪 - 放盒到倉儲
	  70000~71080 : B爪單爪 - 放盒到倉儲
	  80000~81000 : 雙爪 - 放盒到倉儲 (支援同倉/不同倉)
	  99000       : 流程完成
*)
METHOD M_STATE_EXECUTING
VAR_INPUT
END_VAR
VAR_INST
    ActionMode       : E_FeedInToWareHouseAction;   // 動作模式 (單爪A/B、雙爪 × 目標倉儲)
	BoxReady_1st     : BOOL;  // 第一個盒子就緒 (A爪用)
	BoxReady_2nd     : BOOL;  // 第二個盒子就緒 (B爪用)
    CarrierReady_1st : BOOL;  // 第一個載具就緒
    CarrierReady_2nd : BOOL;  // 第二個載具就緒
    uiPickUpBothStep : UINT;  // 雙爪取盒子步驟
    uiPlaceBothStep  : UINT;  // 雙爪放盒子步驟
    ClampA_WareHouseCoordinates : ST_WareHouseCoordinates;  // A爪倉儲目標座標 (Layer/Slide)
    ClampB_WareHouseCoordinates : ST_WareHouseCoordinates;  // B爪倉儲目標座標 (Layer/Slide)
END_VAR
// Set status busy
Busy := TRUE;

// ============================================================
// Step 切換 → Timer 完整歸零
// 解決 tonTimeOut.IN 殘留 TRUE 造成跨 step 累計不歸零
// 每個 step 只要呼叫 tonTimeOut(IN:=TRUE, PT:=...) 啟動計時,
// step 切換瞬間 (uiExecutingStep <> uiExecutingStep_Last) 會被此區塊歸零
// ============================================================
IF uiExecutingStep <> uiExecutingStep_Last THEN
	tonTimeOut(IN := FALSE);
	uiExecutingStep_Last := uiExecutingStep;
END_IF

// Stop 信號: 暫停 timeout 計時 (不歸零, 解除後從停止時間繼續)
IF THIS^.Stop THEN
	tonTimeOut(IN := FALSE);
END_IF

CASE uiExecutingStep OF
    0: // 初始化變數
	// 非自動模式直接報錯 (避免軸控衝突)
	IF GVL_Machine.PackTags[UnitNo.Storage].Status.UnitModeCurrent <> E_UnitMode.Auto THEN
		strStatus := 'FB_FeedInRoundBeltBoxToWareHouse Step 0: Not in Auto mode';
		_UniqueErrorCode := 'E_NOT_AUTO_MODE';
		_Error := TRUE;
	ELSE
        ActionMode       := E_FeedInToWareHouseAction.Undefined;
        CarrierReady_1st := FALSE;
        CarrierReady_2nd := FALSE;
        uiPickUpBothStep := 0;
        uiPlaceBothStep  := 0;
		BoxReady_1st := FALSE;
		BoxReady_2nd := FALSE;
        // 確認命令是否正確 (至少一個爪有 Work)
        IF M_CheckCommand() THEN
            uiExecutingStep := 10;
		ELSE
			strStatus := M_FormatManagedStatus(
				AlarmId := GVL_ErrorCode.GC_ALARM_STO_FEEDIN_RB_TO_WH,
				InnerMessage := GVL_ErrorCode.GC_MSG_0161);
			Status := strStatus;
			Error := TRUE;
			_Error := TRUE;
        END_IF
	END_IF
    10: // 確認各元件就緒
        IF M_CheckUnitsReady() THEN
            uiExecutingStep := 20;
        END_IF
    20: // 確認各元件未忙碌
        IF M_CheckUnitsNotBusy() THEN
            uiExecutingStep := 1000;
        END_IF
    1000: /// 動作模式改為直接判斷 Behavior 決定取盒路徑
        //ActionMode      := M_SelectActionMode();
        uiExecutingStep := 1100;
    1100: // 取得圓帶控制權 (安全卡控：手臂進入圓帶區域，圓帶不可移動)
		DAS_CoreSys.MachineControl.fbAllocateArea.M_GetRoundBeltAccess(ControlAccess := E_RoundBeltControlAccess.FanucRobot);
        // 依動作模式跳轉對應步驟 (直接判斷工作旗標，相容所有 PlaceArea 目的地)
		IF info.ClampA_Setting.Behavior = E_ClampWork.Work AND info.ClampB_Setting.Behavior <> E_ClampWork.Work THEN
			uiExecutingStep := 10000;  // A爪單爪取盒
		ELSIF info.ClampA_Setting.Behavior <> E_ClampWork.Work AND info.ClampB_Setting.Behavior = E_ClampWork.Work THEN
			uiExecutingStep := 20000;  // B爪單爪取盒
		ELSIF info.ClampA_Setting.Behavior = E_ClampWork.Work AND info.ClampB_Setting.Behavior = E_ClampWork.Work THEN
			uiExecutingStep := 30000;  // 雙爪取盒
		ELSE
			_Abort := TRUE;
			strStatus := 'FB_FeedInRoundBeltBoxToWareHouse Step 1100: Invalid Clamp Work Behavior';
			Error := TRUE;
			uiResumeStep := 1100;
		END_IF

{region '第一階段：從圓帶取盒'}
	//=====================================================================
	// 第一階段：從圓帶取盒 (Pick from RoundBelt)
	//=====================================================================

    10000: // A爪單爪 - 移動圓帶到目標站位 (照抄 V2 step 61000 模式)
		DAS_CoreSys.MachineControl.fbAllocateArea.M_GetRoundBeltAccess(ControlAccess := E_RoundBeltControlAccess.FanucRobot);
		DAS_CoreSys.MachineControl.fbAllocateArea.M_StartReloadRoundBeltAtion(ReloadStation := info.ClampA_Setting.RoundBeltSetting.Station);
		IF RoundBelt.xDone AND arAxisCtrl_gb[AxisNo.RoundBelt].Admin.Axis.Status.NotMoving THEN
			DAS_CoreSys.MachineControl.fbAllocateArea.M_ResetReloadRoundBeltAction();
			CarrierReady_1st := TRUE;
			uiExecutingStep := 10010;
		END_IF
		IF RoundBelt.xError THEN
			_Error := TRUE;
			DAS_CoreSys.MachineControl.fbAllocateArea.M_ResetReloadRoundBeltAction();
			strStatus := M_FormatManagedStatus(
				AlarmId := GVL_ErrorCode.GC_ALARM_STO_FEEDIN_RB_TO_WH,
				InnerMessage := GVL_ErrorCode.GC_MSG_0130);
			Status := strStatus;
			Error := TRUE;
		END_IF
	10010: // A爪從圓帶取盒 (使用 PickBoxFromRoundBelt，與 V2 MoveBoxToRoundBelt 對稱)
		IF NOT Robot._DI1.Done THEN
			Robot.M_StartPickBoxFromRoundBelt_ClampA(
				CarrierSelect := info.ClampA_Setting.RoundBeltSetting.ReloadCarrier,
				A2_Sensor     := A2_Sensor,
				A3_Sensor     := A3_Sensor,
				RoundBeltSafe := CarrierReady_1st);
			_AClampDoingWork := TRUE;
			tonTimeOut(IN := TRUE, PT := T#120S);
			IF tonTimeOut.Q THEN
				uiResumeStep := 10010;
				_Abort := TRUE;
				strStatus := M_FormatManagedStatus(
					AlarmId := GVL_ErrorCode.GC_ALARM_STO_FEEDIN_RB_TO_WH,
					InnerMessage := GVL_ErrorCode.GC_MSG_0095);
				Status := strStatus;
				Error := TRUE;
			END_IF
		ELSE
			uiExecutingStep := 10080;
		END_IF
		IF Robot.Error THEN
			uiResumeStep := 10010;
			strStatus := CONCAT('Pick from RoundBelt ClampA Error: ', Robot.ErrMsg);
			Status := strStatus;
			Error := TRUE;
			_Abort := TRUE;
		END_IF
    10080: // A爪取盒完成，釋放圓帶控制權，清除手臂命令，依目的地跳到對應放盒階段
		DAS_CoreSys.MachineControl.fbAllocateArea.M_ResetReloadRoundBeltAction();
		DAS_CoreSys.MachineControl.fbAllocateArea.M_ReleaseRoundBeltAccess(ControlAccess := E_RoundBeltControlAccess.FanucRobot);
        Robot.M_ResetAllCommand();
        IF NOT Robot._DI1.Done THEN
			// 分流: WareHouse → 60000, PullOut → 65000
			IF info.ClampA_Setting.PlaceArea = E_FeedInToWareHouse_PlaceArea.PullOutInner
			OR info.ClampA_Setting.PlaceArea = E_FeedInToWareHouse_PlaceArea.PullOutOuter THEN
				uiExecutingStep := 65000;	// PullOut 放盒
			ELSE
				uiExecutingStep := 60000;	// WareHouse 放盒
			END_IF
        END_IF

    20000: // B爪單爪 - 移動圓帶到目標站位 (照抄 V2 模式)
		DAS_CoreSys.MachineControl.fbAllocateArea.M_GetRoundBeltAccess(ControlAccess := E_RoundBeltControlAccess.FanucRobot);
		DAS_CoreSys.MachineControl.fbAllocateArea.M_StartReloadRoundBeltAtion(ReloadStation := info.ClampB_Setting.RoundBeltSetting.Station);
		IF RoundBelt.xDone AND arAxisCtrl_gb[AxisNo.RoundBelt].Admin.Axis.Status.NotMoving THEN
			DAS_CoreSys.MachineControl.fbAllocateArea.M_ResetReloadRoundBeltAction();
			CarrierReady_2nd := TRUE;
			uiExecutingStep := 20010;
		END_IF
		IF RoundBelt.xError THEN
			_Error := TRUE;
			DAS_CoreSys.MachineControl.fbAllocateArea.M_ResetReloadRoundBeltAction();
			strStatus := M_FormatManagedStatus(
				AlarmId := GVL_ErrorCode.GC_ALARM_STO_FEEDIN_RB_TO_WH,
				InnerMessage := GVL_ErrorCode.GC_MSG_0130);
			Status := strStatus;
			Error := TRUE;
		END_IF
	20010: // B爪從圓帶取盒 (使用 PickBoxFromRoundBelt)
		IF NOT Robot._DI1.Done THEN
			Robot.M_StartPickBoxFromRoundBelt_ClampB(
				CarrierSelect := info.ClampB_Setting.RoundBeltSetting.ReloadCarrier,
				A2_Sensor     := A2_Sensor,
				A3_Sensor     := A3_Sensor,
				RoundBeltSafe := CarrierReady_2nd);
			_BClampDoingWork := TRUE;
			tonTimeOut(IN := TRUE, PT := T#120S);
			IF tonTimeOut.Q THEN
				uiResumeStep := 20010;
				_Abort := TRUE;
				strStatus := M_FormatManagedStatus(
					AlarmId := GVL_ErrorCode.GC_ALARM_STO_FEEDIN_RB_TO_WH,
					InnerMessage := GVL_ErrorCode.GC_MSG_0095);
				Status := strStatus;
				Error := TRUE;
			END_IF
		ELSE
			uiExecutingStep := 20080;
		END_IF
		IF Robot.Error THEN
			uiResumeStep := 20010;
			strStatus := CONCAT('Pick from RoundBelt ClampB Error: ', Robot.ErrMsg);
			Status := strStatus;
			Error := TRUE;
			_Abort := TRUE;
		END_IF
    20080: // B爪取盒完成，釋放圓帶控制權，清除手臂命令，依目的地跳到對應放盒階段
		DAS_CoreSys.MachineControl.fbAllocateArea.M_ResetReloadRoundBeltAction();
		DAS_CoreSys.MachineControl.fbAllocateArea.M_ReleaseRoundBeltAccess(ControlAccess := E_RoundBeltControlAccess.FanucRobot);
        Robot.M_ResetAllCommand();
        IF NOT Robot._DI1.Done THEN
			// 分流: WareHouse → 70000, PullOut → 75000
			IF info.ClampB_Setting.PlaceArea = E_FeedInToWareHouse_PlaceArea.PullOutInner
			OR info.ClampB_Setting.PlaceArea = E_FeedInToWareHouse_PlaceArea.PullOutOuter THEN
				uiExecutingStep := 75000;	// PullOut 放盒
			ELSE
				uiExecutingStep := 70000;	// WareHouse 放盒
			END_IF
        END_IF

    30000: // 雙爪取盒 - 先移動圓帶到 A爪站位 (照抄 V2 模式)
		DAS_CoreSys.MachineControl.fbAllocateArea.M_GetRoundBeltAccess(ControlAccess := E_RoundBeltControlAccess.FanucRobot);
		DAS_CoreSys.MachineControl.fbAllocateArea.M_StartReloadRoundBeltAtion(ReloadStation := info.ClampA_Setting.RoundBeltSetting.Station);
		IF RoundBelt.xDone AND arAxisCtrl_gb[AxisNo.RoundBelt].Admin.Axis.Status.NotMoving THEN
			DAS_CoreSys.MachineControl.fbAllocateArea.M_ResetReloadRoundBeltAction();
			CarrierReady_1st := TRUE;
			uiExecutingStep := 30010;
		END_IF
		IF RoundBelt.xError THEN
			_Error := TRUE;
			//DAS_CoreSys.MachineControl.fbAllocateArea.M_ResetReloadRoundBeltAction();
			strStatus := M_FormatManagedStatus(
				AlarmId := GVL_ErrorCode.GC_ALARM_STO_FEEDIN_RB_TO_WH,
				InnerMessage := GVL_ErrorCode.GC_MSG_0130);
			Status := strStatus;
			Error := TRUE;
		END_IF
	30010: // 雙爪 A爪從圓帶取盒 (使用 PickBoxFromRoundBelt)
		IF NOT Robot._DI1.Done THEN
			Robot.M_StartPickBoxFromRoundBelt_ClampA(
				CarrierSelect := info.ClampA_Setting.RoundBeltSetting.ReloadCarrier,
				A2_Sensor     := A2_Sensor,
				A3_Sensor     := A3_Sensor,
				RoundBeltSafe := CarrierReady_1st);
			_AClampDoingWork := TRUE;
			tonTimeOut(IN := TRUE, PT := T#120S);
			IF tonTimeOut.Q THEN
				uiResumeStep := 30010;
				_Abort := TRUE;
				strStatus := M_FormatManagedStatus(
					AlarmId := GVL_ErrorCode.GC_ALARM_STO_FEEDIN_RB_TO_WH,
					InnerMessage := GVL_ErrorCode.GC_MSG_0093);
				Status := strStatus;
				Error := TRUE;
			END_IF
		ELSE
			uiExecutingStep := 30080;
		END_IF
		IF Robot.Error THEN
			uiResumeStep := 30010;
			strStatus := CONCAT('Pick from RoundBelt ClampA Error: ', Robot.ErrMsg);
			Status := strStatus;
			Error := TRUE;
			_Abort := TRUE;
		END_IF
	30080: // A爪取盒完成，清除手臂命令，準備 B爪取盒 (同站/不同站都重新移動圓帶)
		Robot.M_ResetAllCommand();
		IF NOT Robot._DI1.Done THEN
			uiExecutingStep := 31000;
		END_IF
	31000: // 移動圓帶到 B爪目標站位 (照抄 V2 模式)
		DAS_CoreSys.MachineControl.fbAllocateArea.M_GetRoundBeltAccess(ControlAccess := E_RoundBeltControlAccess.FanucRobot);
		DAS_CoreSys.MachineControl.fbAllocateArea.M_StartReloadRoundBeltAtion(ReloadStation := info.ClampB_Setting.RoundBeltSetting.Station);
		IF RoundBelt.xDone AND arAxisCtrl_gb[AxisNo.RoundBelt].Admin.Axis.Status.NotMoving THEN
			DAS_CoreSys.MachineControl.fbAllocateArea.M_ResetReloadRoundBeltAction();
			CarrierReady_2nd := TRUE;
			uiExecutingStep := 31010;
		END_IF
		IF RoundBelt.xError THEN
			_Error := TRUE;
			DAS_CoreSys.MachineControl.fbAllocateArea.M_ResetReloadRoundBeltAction();
			strStatus := M_FormatManagedStatus(
				AlarmId := GVL_ErrorCode.GC_ALARM_STO_FEEDIN_RB_TO_WH,
				InnerMessage := GVL_ErrorCode.GC_MSG_0130);
			Status := strStatus;
			Error := TRUE;
		END_IF
	31010: // 雙爪 B爪從圓帶取盒 (使用 PickBoxFromRoundBelt)
		IF NOT Robot._DI1.Done THEN
			Robot.M_StartPickBoxFromRoundBelt_ClampB(
				CarrierSelect := info.ClampB_Setting.RoundBeltSetting.ReloadCarrier,
				A2_Sensor     := A2_Sensor,
				A3_Sensor     := A3_Sensor,
				RoundBeltSafe := CarrierReady_2nd);
			_BClampDoingWork := TRUE;
			tonTimeOut(IN := TRUE, PT := T#120S);
			IF tonTimeOut.Q THEN
				uiResumeStep := 31010;
				_Abort := TRUE;
				strStatus := M_FormatManagedStatus(
					AlarmId := GVL_ErrorCode.GC_ALARM_STO_FEEDIN_RB_TO_WH,
					InnerMessage := GVL_ErrorCode.GC_MSG_0094);
				Status := strStatus;
				Error := TRUE;
			END_IF
		ELSE
			uiExecutingStep := 31080;
		END_IF
		IF Robot.Error THEN
			uiResumeStep := 31010;
			strStatus := CONCAT('Pick from RoundBelt ClampB Error: ', Robot.ErrMsg);
			Status := strStatus;
			Error := TRUE;
			_Abort := TRUE;
		END_IF
	31080: // 雙爪取盒完成，釋放圓帶控制權，依 destination 分流
		DAS_CoreSys.MachineControl.fbAllocateArea.M_ResetReloadRoundBeltAction();
		DAS_CoreSys.MachineControl.fbAllocateArea.M_ReleaseRoundBeltAccess(ControlAccess := E_RoundBeltControlAccess.FanucRobot);
		Robot.M_ResetAllCommand();
		IF NOT Robot._DI1.Done THEN
			// 雙爪都是 WareHouse → 走 80000 (有同/不同倉的同步優化路徑)
			// 任一爪有 PullOut → 走 86000 sequential dispatch (先 A 後 B)
			IF (info.ClampA_Setting.PlaceArea = E_FeedInToWareHouse_PlaceArea.WareHouseA
			 OR info.ClampA_Setting.PlaceArea = E_FeedInToWareHouse_PlaceArea.WareHouseB)
			AND (info.ClampB_Setting.PlaceArea = E_FeedInToWareHouse_PlaceArea.WareHouseA
			 OR info.ClampB_Setting.PlaceArea = E_FeedInToWareHouse_PlaceArea.WareHouseB)
			THEN
				uiExecutingStep := 80000;
			ELSE
				uiExecutingStep := 86000;	// dual sequential (含 PullOut 或 mixed)
			END_IF
		END_IF
{endregion}

{region '第二階段：放盒到倉儲'}
	//=====================================================================
	// 第二階段：放盒到倉儲 (Place to WareHouse)
	//=====================================================================

    60000: // A爪單爪放盒 - 清除手臂命令，確認手臂閒置
        Robot.M_ResetAllCommand();
        // 確認手臂沒有在執行其他動作
        IF NOT Robot._di1.Done AND
            NOT (Robot._DI1.AbsMoveA OR
            Robot._DI1.AbsMoveB OR
            Robot._DI1.WarehouseA OR
            Robot._DI1.WarehouseB) THEN
            uiExecutingStep := 61000;
        END_IF
    61000: // A爪放盒到倉儲 (照抄 V2 模式：同時驅動倉儲 FeedIn + Robot Place，光電板 sensor 確認軌道空)
		ClampA_WareHouseCoordinates := info.ClampA_Setting.WareHouseSetting;
        IF NOT Robot._DI1.Done THEN
            IF info.ClampA_Setting.PlaceArea = E_FeedInToWareHouse_PlaceArea.WareHouseA THEN
				WareHouse.M_StartFeedInBox(WareHouseSelect := E_WareHouse.WareHouseA, WarehouseCoordinates := ClampA_WareHouseCoordinates);
				IF WareHouse.bFeedInBox_Completed THEN
					BoxReady_1st := TRUE;
				END_IF
                Robot.M_StartWareHousePlaceBox_ClampA(
                    WareHouseSelect := E_WareHouse.WareHouseA,
                    Info            := ClampA_WareHouseCoordinates,
                    BoxReady_1st    := BoxReady_1st);
            ELSIF info.ClampA_Setting.PlaceArea = E_FeedInToWareHouse_PlaceArea.WareHouseB THEN
				WareHouse.M_StartFeedInBox(WareHouseSelect := E_WareHouse.WareHouseB, WarehouseCoordinates := ClampA_WareHouseCoordinates);
				IF WareHouse.bFeedInBox_Completed THEN
					BoxReady_1st := TRUE;
				END_IF
                Robot.M_StartWareHousePlaceBox_ClampA(
                    WareHouseSelect := E_WareHouse.WareHouseB,
                    Info            := ClampA_WareHouseCoordinates,
                    BoxReady_1st    := BoxReady_1st);
            END_IF
			tonTimeOut(IN := TRUE, PT := T#120S);
			IF tonTimeOut.Q THEN
				uiResumeStep := 61000;
				_Abort := TRUE;
				strStatus := M_FormatManagedStatus(
					AlarmId := GVL_ErrorCode.GC_ALARM_STO_FEEDIN_RB_TO_WH,
					InnerMessage := GVL_ErrorCode.GC_MSG_0098);
				Status := strStatus;
				Error := TRUE;
			END_IF
        ELSE
            uiExecutingStep := 61080;
        END_IF
    61080: // A爪放盒完成，設 AClampMoveDone，清除手臂命令
		IF NOT AClampMoveDone THEN
			AClampMoveDone := TRUE;
			M_AppendActionRecord_ClampA();
		END_IF
        Robot.M_ResetAllCommand();
        IF NOT Robot._DI1.Done THEN
            uiExecutingStep := 62000;
        END_IF
	62000: // 等待倉儲 FeedIn 完成 → Reset → 訊號關
		IF WareHouse.bFeedInBox_Completed THEN
			WareHouse.M_ResetFeedInBox();
			uiExecutingStep := 62010;
		END_IF
	62010:
		IF NOT WareHouse.bFeedInBox_Completed THEN
			uiExecutingStep := 99000;
		END_IF

    70000: // B爪單爪放盒 - 清除手臂命令，確認手臂閒置
        Robot.M_ResetAllCommand();
        IF NOT Robot._di1.Done AND
            NOT (Robot._DI1.AbsMoveA OR
            Robot._DI1.AbsMoveB OR
            Robot._DI1.WarehouseA OR
            Robot._DI1.WarehouseB) THEN
            uiExecutingStep := 71000;
        END_IF
    71000: // B爪放盒到倉儲 (照抄 V2 模式：同時驅動倉儲 FeedIn + Robot Place)
		ClampB_WareHouseCoordinates := info.ClampB_Setting.WareHouseSetting;
        IF NOT Robot._DI1.Done THEN
            IF info.ClampB_Setting.PlaceArea = E_FeedInToWareHouse_PlaceArea.WareHouseA THEN
				WareHouse.M_StartFeedInBox(WareHouseSelect := E_WareHouse.WareHouseA, WarehouseCoordinates := ClampB_WareHouseCoordinates);
				IF WareHouse.bFeedInBox_Completed THEN
					BoxReady_2nd := TRUE;
				END_IF
                Robot.M_StartWareHousePlaceBox_ClampB(
                    WareHouseSelect := E_WareHouse.WareHouseA,
                    Info            := ClampB_WareHouseCoordinates,
                    BoxReady_2nd    := BoxReady_2nd);
            ELSIF info.ClampB_Setting.PlaceArea = E_FeedInToWareHouse_PlaceArea.WareHouseB THEN
				WareHouse.M_StartFeedInBox(WareHouseSelect := E_WareHouse.WareHouseB, WarehouseCoordinates := ClampB_WareHouseCoordinates);
				IF WareHouse.bFeedInBox_Completed THEN
					BoxReady_2nd := TRUE;
				END_IF
                Robot.M_StartWareHousePlaceBox_ClampB(
                    WareHouseSelect := E_WareHouse.WareHouseB,
                    Info            := ClampB_WareHouseCoordinates,
                    BoxReady_2nd    := BoxReady_2nd);
            END_IF
			tonTimeOut(IN := TRUE, PT := T#120S);
			IF tonTimeOut.Q THEN
				uiResumeStep := 71000;
				_Abort := TRUE;
				strStatus := M_FormatManagedStatus(
					AlarmId := GVL_ErrorCode.GC_ALARM_STO_FEEDIN_RB_TO_WH,
					InnerMessage := GVL_ErrorCode.GC_MSG_0098);
				Status := strStatus;
				Error := TRUE;
			END_IF
        ELSE
            uiExecutingStep := 71080;
        END_IF
    71080: // B爪放盒完成，設 BClampMoveDone，清除手臂命令
		IF NOT BClampMoveDone THEN
			BClampMoveDone := TRUE;
			M_AppendActionRecord_ClampB();
		END_IF
        Robot.M_ResetAllCommand();
        IF NOT Robot._DI1.Done THEN
            uiExecutingStep := 72000;
        END_IF
	72000: // 等待倉儲 FeedIn 完成 → Reset → 訊號關
		IF WareHouse.bFeedInBox_Completed THEN
			WareHouse.M_ResetFeedInBox();
			uiExecutingStep := 72010;
		END_IF
	72010:
		IF NOT WareHouse.bFeedInBox_Completed THEN
			uiExecutingStep := 99000;
		END_IF

	//=====================================================================
	// 第二階段 (PullOut 變體): 放盒到 PullOutConveyor (僅單爪 MVP)
	// PlaceArea = PullOutInner (I3_Slide, Address=1, 機台內側/左) / PullOutOuter (I4_Slide, Address=2, 機台外側/右)
	// 使用 Robot.M_StartRobotAbsMove(Area=PullOutConveyor, GetBox=FALSE)
	// 走 fbAllocateArea 共用入口 (跟 FB_RobotRegionMove_PullOutConveyor 同 pattern)
	//=====================================================================

	65000: // A爪 PullOut 放盒 - 清手臂命令、確認手臂閒置、取得 PullOut 控制權
		Robot.M_ResetAllCommand();
		IF NOT Robot._DI1.Done AND
			NOT (Robot._DI1.AbsMoveA OR Robot._DI1.AbsMoveB OR
				 Robot._DI1.WarehouseA OR Robot._DI1.WarehouseB) THEN
			DAS_CoreSys.MachineControl.fbAllocateArea.M_GetPulloutAccess(ControlAccess := E_RoundBeltControlAccess.FanucRobot);
			uiExecutingStep := 65010;
		END_IF

